LIN {X 0,Y 184.032,Z 367.437,A -85,B 0,C 180,E1 -22186.576,E2 -22186.576} C_VEL
LIN {X 0,Y 183.356,Z 367.135,A -85,B 0,C 180,E1 -22190.049,E2 -22190.049} C_VEL
LIN {X 0,Y 183.093,Z 365.736,A -85,B 0,C 180,E1 -22193.714,E2 -22193.714} C_VEL
LIN {X 0,Y 183.399,Z 363.047,A -85,B 0,C 180,E1 -22197.555,E2 -22197.555} C_VEL
LIN {X 0,Y 184.194,Z 359.068,A -85,B 0,C 180,E1 -22201.35,E2 -22201.35} C_VEL
LIN {X 0,Y 185.42,Z 353.009,A -85,B 0,C 180,E1 -22205.459,E2 -22205.459} C_VEL
LIN {X 0,Y 186.983,Z 346.449,A -85,B 0,C 180,E1 -22208.832,E2 -22208.832} C_VEL
LIN {X 0,Y 188.948,Z 338.257,A -85,B 0,C 180,E1 -22212.13,E2 -22212.13} C_VEL
LIN {X 0,Y 191.271,Z 328.831,A -85,B 0,C 180,E1 -22215.096,E2 -22215.096} C_VEL
LIN {X 0,Y 193.258,Z 319.749,A -85,B 0,C 180,E1 -22217.397,E2 -22217.397} C_VEL
LIN {X 0,Y 195.527,Z 308.58,A -85,B 0,C 180,E1 -22219.647,E2 -22219.647} C_VEL
LIN {X 0,Y 197.745,Z 296.151,A -85,B 0,C 180,E1 -22221.57,E2 -22221.57} C_VEL
LIN {X 0,Y 199.324,Z 284.381,A -85,B 0,C 180,E1 -22222.968,E2 -22222.968} C_VEL
LIN {X 0,Y 200.748,Z 270.755,A -85,B 0,C 180,E1 -22224.108,E2 -22224.108} C_VEL
LIN {X 0,Y 201.714,Z 257.362,A -85,B 0,C 180,E1 -22224.816,E2 -22224.816} C_VEL
LIN {X 0,Y 204.371,Z 205.343,A -85,B 0,C 180,E1 -22226.746,E2 -22226.746} C_VEL
LIN {X 0,Y 197.795,Z 189.738,A -85,B 0,C 180,E1 -22228.409,E2 -22228.409} C_VEL
LIN {X 0,Y 187.977,Z 169.046,A -85,B 0,C 180,E1 -22231.002,E2 -22231.002} C_VEL
LIN {X 0,Y 186.53,Z 166.516,A -85,B 0,C 180,E1 -22231.384,E2 -22231.384} C_VEL
LIN {X 0,Y 186.263,Z 165.286,A -85,B 0,C 180,E1 -22231.555,E2 -22231.555} C_VEL
LIN {X 0,Y 185.974,Z 165.321,A -85,B 0,C 180,E1 -22238.694,E2 -22238.694} C_VEL
LIN {X 0,Y 185.717,Z 165.352,A -85,B 0,C 180,E1 -22243.124,E2 -22243.124} C_VEL
LIN {X 0,Y 185.656,Z 165.356,A -85,B 0,C 180,E1 -22247.628,E2 -22247.628} C_VEL
LIN {X 0,Y 185.574,Z 165.367,A -85,B 0,C 180,E1 -22252.254,E2 -22252.254} C_VEL
LIN {X 0,Y 185.56,Z 165.368,A -85,B 0,C 180,E1 -22257.032,E2 -22257.032} C_VEL
LIN {X 0,Y 185.579,Z 165.367,A -85,B 0,C 180,E1 -22259.493,E2 -22259.493} C_VEL
LIN {X 0,Y 185.499,Z 165.377,A -85,B 0,C 180,E1 -22264.632,E2 -22264.632} C_VEL
LIN {X 0,Y 185.505,Z 165.377,A -85,B 0,C 180,E1 -22267.313,E2 -22267.313} C_VEL
LIN {X 0,Y 185.47,Z 165.369,A -85,B 0,C 180,E1 -22270.725,E2 -22270.725} C_VEL
LIN {X 0,Y 185.459,Z 165.384,A -85,B 0,C 180,E1 -22276.055,E2 -22276.055} C_VEL
LIN {X 0,Y 185.487,Z 165.365,A -85,B 0,C 180,E1 -22279.901,E2 -22279.901} C_VEL
LIN {X 0,Y 185.543,Z 165.368,A -85,B 0,C 180,E1 -22282.696,E2 -22282.696} C_VEL
LIN {X 0,Y 185.54,Z 165.366,A -85,B 0,C 180,E1 -22287.975,E2 -22287.975} C_VEL
LIN {X 0,Y 185.58,Z 165.348,A -85,B 0,C 180,E1 -22290.577,E2 -22290.577} C_VEL
LIN {X 0,Y 185.579,Z 165.367,A -85,B 0,C 180,E1 -22295.382,E2 -22295.382} C_VEL
LIN {X 0,Y 185.673,Z 165.341,A -85,B 0,C 180,E1 -22301.135,E2 -22301.135} C_VEL
LIN {X 0,Y 185.724,Z 165.342,A -85,B 0,C 180,E1 -22304.64,E2 -22304.64} C_VEL
LIN {X 0,Y 185.924,Z 165.323,A -85,B 0,C 180,E1 -22309.359,E2 -22309.359} C_VEL
LIN {X 0,Y 185.961,Z 165.303,A -85,B 0,C 180,E1 -22313.49,E2 -22313.49} C_VEL
LIN {X 0,Y 186.208,Z 165.286,A -85,B 0,C 180,E1 -22317.837,E2 -22317.837} C_VEL
LIN {X 0,Y 186.407,Z 165.26,A -85,B 0,C 180,E1 -22320,E2 -22320} C_VEL
LIN {X 0,Y 185.923,Z 165.31,A -85,B 0,C 180,E1 -22324.336,E2 -22324.336} C_VEL
LIN {X 0,Y 186.009,Z 165.314,A -85,B 0,C 180,E1 -22328.693,E2 -22328.693} C_VEL
LIN {X 0,Y 185.765,Z 165.335,A -85,B 0,C 180,E1 -22333.121,E2 -22333.121} C_VEL
LIN {X 0,Y 185.69,Z 165.353,A -85,B 0,C 180,E1 -22337.625,E2 -22337.625} C_VEL
LIN {X 0,Y 185.579,Z 165.366,A -85,B 0,C 180,E1 -22342.254,E2 -22342.254} C_VEL
LIN {X 0,Y 185.561,Z 165.365,A -85,B 0,C 180,E1 -22347.033,E2 -22347.033} C_VEL
LIN {X 0,Y 185.58,Z 165.369,A -85,B 0,C 180,E1 -22349.493,E2 -22349.493} C_VEL
LIN {X 0,Y 185.52,Z 165.377,A -85,B 0,C 180,E1 -22354.628,E2 -22354.628} C_VEL
LIN {X 0,Y 185.545,Z 165.372,A -85,B 0,C 180,E1 -22357.304,E2 -22357.304} C_VEL
LIN {X 0,Y 185.504,Z 165.379,A -85,B 0,C 180,E1 -22360.737,E2 -22360.737} C_VEL
LIN {X 0,Y 185.519,Z 165.377,A -85,B 0,C 180,E1 -22366.037,E2 -22366.037} C_VEL
LIN {X 0,Y 185.542,Z 165.525,A -85,B 0,C 180,E1 -22366.821,E2 -22366.821} C_VEL
LIN {X 0,Y 187.738,Z 174.486,A -85,B 0,C 180,E1 -22371.323,E2 -22371.323} C_VEL
LIN {X 0,Y 196.018,Z 195.049,A -85,B 0,C 180,E1 -22373.668,E2 -22373.668} C_VEL
LIN {X 0,Y 199.664,Z 205.529,A -85,B 0,C 180,E1 -22374.697,E2 -22374.697} C_VEL
LIN {X 0,Y 202.857,Z 235.414,A -85,B 0,C 180,E1 -22376.487,E2 -22376.487} C_VEL
LIN {X 0,Y 202.626,Z 245.83,A -85,B 0,C 180,E1 -22376.916,E2 -22376.916} C_VEL
LIN {X 0,Y 202.405,Z 251.4,A -85,B 0,C 180,E1 -22377.132,E2 -22377.132} C_VEL
LIN {X 0,Y 201.656,Z 257.229,A -85,B 0,C 180,E1 -22377.285,E2 -22377.285} C_VEL
LIN {X 0,Y 198.546,Z 266.659,A -85,B 0,C 180,E1 -22377.284,E2 -22377.284} C_VEL
LIN {X 0,Y 195.295,Z 276.077,A -85,B 0,C 180,E1 -22377.291,E2 -22377.291} C_VEL
LIN {X 0,Y 194.336,Z 281.893,A -85,B 0,C 180,E1 -22377.468,E2 -22377.468} C_VEL
LIN {X 0,Y 193.33,Z 293.632,A -85,B 0,C 180,E1 -22378.19,E2 -22378.19} C_VEL
LIN {X 0,Y 191.752,Z 305.726,A -85,B 0,C 180,E1 -22379.281,E2 -22379.281} C_VEL
LIN {X 0,Y 189.786,Z 316.758,A -85,B 0,C 180,E1 -22380.616,E2 -22380.616} C_VEL
LIN {X 0,Y 187.216,Z 329.252,A -85,B 0,C 180,E1 -22382.622,E2 -22382.622} C_VEL
LIN {X 0,Y 184.684,Z 340.28,A -85,B 0,C 180,E1 -22384.954,E2 -22384.954} C_VEL
LIN {X 0,Y 182.202,Z 350.699,A -85,B 0,C 180,E1 -22387.782,E2 -22387.782} C_VEL
LIN {X 0,Y 180.484,Z 357.527,A -85,B 0,C 180,E1 -22390.079,E2 -22390.079} C_VEL
LIN {X 0,Y 178.673,Z 365.629,A -85,B 0,C 180,E1 -22393.431,E2 -22393.431} C_VEL
LIN {X 0,Y 177.448,Z 371.066,A -85,B 0,C 180,E1 -22396.253,E2 -22396.253} C_VEL
LIN {X 0,Y 176.647,Z 376.382,A -85,B 0,C 180,E1 -22399.686,E2 -22399.686} C_VEL
LIN {X 0,Y 176.33,Z 380.466,A -85,B 0,C 180,E1 -22403.133,E2 -22403.133} C_VEL
LIN {X 0,Y 176.351,Z 382.551,A -85,B 0,C 180,E1 -22405.428,E2 -22405.428} C_VEL
LIN {X 0,Y 176.404,Z 384.172,A -85,B 0,C 180,E1 -22407.717,E2 -22407.717} C_VEL
LIN {X 0,Y 176.485,Z 385.363,A -85,B 0,C 180,E1 -22410,E2 -22410} C_VEL
LIN {X 0,Y 176.309,Z 386.103,A -85,B 0,C 180,E1 -22412.284,E2 -22412.284} C_VEL
LIN {X 0,Y 176.145,Z 386.398,A -85,B 0,C 180,E1 -22414.577,E2 -22414.577} C_VEL
LIN {X 0,Y 176.371,Z 385.833,A -85,B 0,C 180,E1 -22419.171,E2 -22419.171} C_VEL
LIN {X 0,Y 176.852,Z 384.98,A -85,B 0,C 180,E1 -22421.461,E2 -22421.461} C_VEL
LIN {X 0,Y 178.535,Z 382.023,A -85,B 0,C 180,E1 -22425.995,E2 -22425.995} C_VEL
LIN {X 0,Y 180.694,Z 378.736,A -85,B 0,C 180,E1 -22429.305,E2 -22429.305} C_VEL
LIN {X 0,Y 183.399,Z 374.424,A -85,B 0,C 180,E1 -22432.532,E2 -22432.532} C_VEL
LIN {X 0,Y 187.159,Z 367.956,A -85,B 0,C 180,E1 -22436.182,E2 -22436.182} C_VEL
LIN {X 0,Y 191.107,Z 360.986,A -85,B 0,C 180,E1 -22439.161,E2 -22439.161} C_VEL
LIN {X 0,Y 195.635,Z 352.395,A -85,B 0,C 180,E1 -22441.997,E2 -22441.997} C_VEL
LIN {X 0,Y 199.979,Z 343.651,A -85,B 0,C 180,E1 -22444.215,E2 -22444.215} C_VEL
LIN {X 0,Y 204.06,Z 334.168,A -85,B 0,C 180,E1 -22446.142,E2 -22446.142} C_VEL
LIN {X 0,Y 208.011,Z 323.894,A -85,B 0,C 180,E1 -22447.762,E2 -22447.762} C_VEL
LIN {X 0,Y 211.57,Z 312.785,A -85,B 0,C 180,E1 -22449.134,E2 -22449.134} C_VEL
LIN {X 0,Y 214.827,Z 300.374,A -85,B 0,C 180,E1 -22450.249,E2 -22450.249} C_VEL
LIN {X 0,Y 217.351,Z 286.914,A -85,B 0,C 180,E1 -22451.126,E2 -22451.126} C_VEL
LIN {X 0,Y 218.947,Z 273.192,A -85,B 0,C 180,E1 -22451.698,E2 -22451.698} C_VEL
LIN {X 0,Y 221.305,Z 243.676,A -85,B 0,C 180,E1 -22452.714,E2 -22452.714} C_VEL
LIN {X 0,Y 220.723,Z 234.505,A -85,B 0,C 180,E1 -22453.502,E2 -22453.502} C_VEL
LIN {X 0,Y 216.604,Z 223.631,A -85,B 0,C 180,E1 -22455.788,E2 -22455.788} C_VEL
LIN {X 0,Y 212.688,Z 215.258,A -85,B 0,C 180,E1 -22458.109,E2 -22458.109} C_VEL
LIN {X 0,Y 209.577,Z 209.321,A -85,B 0,C 180,E1 -22460.11,E2 -22460.11} C_VEL
LIN {X 0,Y 207.305,Z 205.119,A -85,B 0,C 180,E1 -22461.75,E2 -22461.75} C_VEL
LIN {X 0,Y 204.342,Z 199.923,A -85,B 0,C 180,E1 -22464.107,E2 -22464.107} C_VEL
LIN {X 0,Y 200.97,Z 194.246,A -85,B 0,C 180,E1 -22467.349,E2 -22467.349} C_VEL
LIN {X 0,Y 196.57,Z 187.167,A -85,B 0,C 180,E1 -22473.357,E2 -22473.357} C_VEL
LIN {X 0,Y 194.473,Z 184.049,A -85,B 0,C 180,E1 -22479.652,E2 -22479.652} C_VEL
LIN {X 0,Y 194.709,Z 184.022,A -85,B 0,C 180,E1 -22485.364,E2 -22485.364} C_VEL
LIN {X 0,Y 196.216,Z 184.626,A -85,B 0,C 180,E1 -22489.292,E2 -22489.292} C_VEL
LIN {X 0,Y 197.724,Z 187.889,A -85,B 0,C 180,E1 -22492.253,E2 -22492.253} C_VEL
LIN {X 0,Y 200.136,Z 189.87,A -85,B 0,C 180,E1 -22495.215,E2 -22495.215} C_VEL
LIN {X 0,Y 200.777,Z 190.672,A -85,B 0,C 180,E1 -22495.922,E2 -22495.922} C_VEL
LIN {X 0,Y 203.022,Z 193.797,A -85,B 0,C 180,E1 -22498.147,E2 -22498.147} C_VEL
LIN {X 0,Y 203.994,Z 195.111,A -85,B 0,C 180,E1 -22499.022,E2 -22499.022} C_VEL
LIN {X 0,Y 206.507,Z 198.84,A -85,B 0,C 180,E1 -22501.071,E2 -22501.071} C_VEL
LIN {X 0,Y 210.473,Z 204.645,A -85,B 0,C 180,E1 -22503.865,E2 -22503.865} C_VEL
LIN {X 0,Y 214.841,Z 211.746,A -85,B 0,C 180,E1 -22506.499,E2 -22506.499} C_VEL
LIN {X 0,Y 219.364,Z 219.717,A -85,B 0,C 180,E1 -22508.927,E2 -22508.927} C_VEL
LIN {X 0,Y 222.627,Z 226.3,A -85,B 0,C 180,E1 -22510.552,E2 -22510.552} C_VEL
LIN {X 0,Y 219.091,Z 267.39,A -85,B 0,C 180,E1 -22511.994,E2 -22511.994} C_VEL
LIN {X 0,Y 217.001,Z 281.249,A -85,B 0,C 180,E1 -22512.82,E2 -22512.82} C_VEL
LIN {X 0,Y 214.473,Z 293.514,A -85,B 0,C 180,E1 -22513.926,E2 -22513.926} C_VEL
LIN {X 0,Y 211.106,Z 305.921,A -85,B 0,C 180,E1 -22515.446,E2 -22515.446} C_VEL
LIN {X 0,Y 207.644,Z 316.071,A -85,B 0,C 180,E1 -22517.03,E2 -22517.03} C_VEL
LIN {X 0,Y 203.566,Z 326.285,A -85,B 0,C 180,E1 -22519.074,E2 -22519.074} C_VEL
LIN {X 0,Y 199.211,Z 335.653,A -85,B 0,C 180,E1 -22521.49,E2 -22521.49} C_VEL
LIN {X 0,Y 194.694,Z 344.181,A -85,B 0,C 180,E1 -22524.314,E2 -22524.314} C_VEL
LIN {X 0,Y 190.253,Z 351.606,A -85,B 0,C 180,E1 -22527.556,E2 -22527.556} C_VEL
LIN {X 0,Y 186.095,Z 357.882,A -85,B 0,C 180,E1 -22531.255,E2 -22531.255} C_VEL
LIN {X 0,Y 183.362,Z 361.587,A -85,B 0,C 180,E1 -22534.231,E2 -22534.231} C_VEL
LIN {X 0,Y 180.342,Z 365.302,A -85,B 0,C 180,E1 -22538.573,E2 -22538.573} C_VEL
LIN {X 0,Y 178.539,Z 367.039,A -85,B 0,C 180,E1 -22542.004,E2 -22542.004} C_VEL
LIN {X 0,Y 177.177,Z 367.836,A -85,B 0,C 180,E1 -22545.56,E2 -22545.56} C_VEL
LIN {X 0,Y 176.375,Z 367.638,A -85,B 0,C 180,E1 -22549.208,E2 -22549.208} C_VEL
LIN {X 0,Y 176.004,Z 366.246,A -85,B 0,C 180,E1 -22553.205,E2 -22553.205} C_VEL
LIN {X 0,Y 176.195,Z 363.867,A -85,B 0,C 180,E1 -22556.891,E2 -22556.891} C_VEL
LIN {X 0,Y 176.985,Z 359.996,A -85,B 0,C 180,E1 -22560.88,E2 -22560.88} C_VEL
LIN {X 0,Y 177.881,Z 355.57,A -85,B 0,C 180,E1 -22564.24,E2 -22564.24} C_VEL
LIN {X 0,Y 179.467,Z 348.824,A -85,B 0,C 180,E1 -22568.16,E2 -22568.16} C_VEL
LIN {X 0,Y 181.225,Z 341.748,A -85,B 0,C 180,E1 -22571.341,E2 -22571.341} C_VEL
LIN {X 0,Y 183.394,Z 333.098,A -85,B 0,C 180,E1 -22574.44,E2 -22574.44} C_VEL
LIN {X 0,Y 185.765,Z 323.252,A -85,B 0,C 180,E1 -22577.242,E2 -22577.242} C_VEL
LIN {X 0,Y 188.293,Z 311.74,A -85,B 0,C 180,E1 -22579.788,E2 -22579.788} C_VEL
LIN {X 0,Y 190.52,Z 300.077,A -85,B 0,C 180,E1 -22581.799,E2 -22581.799} C_VEL
LIN {X 0,Y 192.302,Z 288.407,A -85,B 0,C 180,E1 -22583.337,E2 -22583.337} C_VEL
LIN {X 0,Y 193.911,Z 274.589,A -85,B 0,C 180,E1 -22584.671,E2 -22584.671} C_VEL
LIN {X 0,Y 195.004,Z 261.627,A -85,B 0,C 180,E1 -22585.478,E2 -22585.478} C_VEL
LIN {X 0,Y 197.86,Z 206.871,A -85,B 0,C 180,E1 -22587.608,E2 -22587.608} C_VEL
LIN {X 0,Y 191.853,Z 192.642,A -85,B 0,C 180,E1 -22589.197,E2 -22589.197} C_VEL
LIN {X 0,Y 182.808,Z 173.416,A -85,B 0,C 180,E1 -22591.711,E2 -22591.711} C_VEL
LIN {X 0,Y 180.157,Z 169.113,A -85,B 0,C 180,E1 -22592.429,E2 -22592.429} C_VEL
LIN {X 0,Y 179.041,Z 166.186,A -85,B 0,C 180,E1 -22592.813,E2 -22592.813} C_VEL
LIN {X 0,Y 178.905,Z 166.204,A -85,B 0,C 180,E1 -22599.041,E2 -22599.041} C_VEL
LIN {X 0,Y 178.644,Z 166.233,A -85,B 0,C 180,E1 -22603.653,E2 -22603.653} C_VEL
LIN {X 0,Y 178.59,Z 166.239,A -85,B 0,C 180,E1 -22609.186,E2 -22609.186} C_VEL
LIN {X 0,Y 178.519,Z 166.247,A -85,B 0,C 180,E1 -22615.114,E2 -22615.114} C_VEL
LIN {X 0,Y 178.523,Z 166.246,A -85,B 0,C 180,E1 -22619.994,E2 -22619.994} C_VEL
LIN {X 0,Y 178.485,Z 166.252,A -85,B 0,C 180,E1 -22624.22,E2 -22624.22} C_VEL
LIN {X 0,Y 178.395,Z 166.258,A -85,B 0,C 180,E1 -22629.075,E2 -22629.075} C_VEL
LIN {X 0,Y 178.397,Z 166.251,A -85,B 0,C 180,E1 -22632.045,E2 -22632.045} C_VEL
LIN {X 0,Y 178.393,Z 166.262,A -85,B 0,C 180,E1 -22635.164,E2 -22635.164} C_VEL
LIN {X 0,Y 178.409,Z 166.252,A -85,B 0,C 180,E1 -22638.457,E2 -22638.457} C_VEL
LIN {X 0,Y 178.463,Z 166.243,A -85,B 0,C 180,E1 -22641.963,E2 -22641.963} C_VEL
LIN {X 0,Y 178.489,Z 166.248,A -85,B 0,C 180,E1 -22646.548,E2 -22646.548} C_VEL
LIN {X 0,Y 178.521,Z 166.229,A -85,B 0,C 180,E1 -22650.008,E2 -22650.008} C_VEL
LIN {X 0,Y 178.519,Z 166.245,A -85,B 0,C 180,E1 -22654.886,E2 -22654.886} C_VEL
LIN {X 0,Y 178.621,Z 166.221,A -85,B 0,C 180,E1 -22660.786,E2 -22660.786} C_VEL
LIN {X 0,Y 178.665,Z 166.218,A -85,B 0,C 180,E1 -22664.017,E2 -22664.017} C_VEL
LIN {X 0,Y 178.861,Z 166.203,A -85,B 0,C 180,E1 -22669.211,E2 -22669.211} C_VEL
LIN {X 0,Y 178.925,Z 166.178,A -85,B 0,C 180,E1 -22673.233,E2 -22673.233} C_VEL
LIN {X 0,Y 179.154,Z 166.165,A -85,B 0,C 180,E1 -22677.752,E2 -22677.752} C_VEL
LIN {X 0,Y 179.37,Z 166.137,A -85,B 0,C 180,E1 -22680,E2 -22680} C_VEL
LIN {X 0,Y 178.871,Z 166.189,A -85,B 0,C 180,E1 -22684.508,E2 -22684.508} C_VEL
LIN {X 0,Y 178.96,Z 166.191,A -85,B 0,C 180,E1 -22689.038,E2 -22689.038} C_VEL
LIN {X 0,Y 178.687,Z 166.219,A -85,B 0,C 180,E1 -22693.65,E2 -22693.65} C_VEL
LIN {X 0,Y 178.649,Z 166.229,A -85,B 0,C 180,E1 -22698.344,E2 -22698.344} C_VEL
LIN {X 0,Y 178.498,Z 166.25,A -85,B 0,C 180,E1 -22703.187,E2 -22703.187} C_VEL
LIN {X 0,Y 178.487,Z 166.25,A -85,B 0,C 180,E1 -22708.198,E2 -22708.198} C_VEL
LIN {X 0,Y 178.48,Z 166.252,A -85,B 0,C 180,E1 -22710.791,E2 -22710.791} C_VEL
LIN {X 0,Y 178.497,Z 166.253,A -85,B 0,C 180,E1 -22714.225,E2 -22714.225} C_VEL
LIN {X 0,Y 178.427,Z 166.258,A -85,B 0,C 180,E1 -22719.067,E2 -22719.067} C_VEL
LIN {X 0,Y 178.433,Z 166.258,A -85,B 0,C 180,E1 -22722.036,E2 -22722.036} C_VEL
LIN {X 0,Y 178.497,Z 166.39,A -85,B 0,C 180,E1 -22725.937,E2 -22725.937} C_VEL
LIN {X 0,Y 180.402,Z 174.103,A -85,B 0,C 180,E1 -22729.974,E2 -22729.974} C_VEL
LIN {X 0,Y 187.223,Z 190.403,A -85,B 0,C 180,E1 -22732.028,E2 -22732.028} C_VEL
LIN {X 0,Y 193.54,Z 207.992,A -85,B 0,C 180,E1 -22733.898,E2 -22733.898} C_VEL
LIN {X 0,Y 196.515,Z 237.335,A -85,B 0,C 180,E1 -22735.695,E2 -22735.695} C_VEL
LIN {X 0,Y 194.646,Z 277.657,A -85,B 0,C 180,E1 -22737.285,E2 -22737.285} C_VEL
LIN {X 0,Y 194.336,Z 281.893,A -85,B 0,C 180,E1 -22737.468,E2 -22737.468} C_VEL
LIN {X 0,Y 193.328,Z 287.66,A -85,B 0,C 180,E1 -22737.702,E2 -22737.702} C_VEL
LIN {X 0,Y 189.715,Z 296.836,A -85,B 0,C 180,E1 -22738.027,E2 -22738.027} C_VEL
LIN {X 0,Y 185.718,Z 305.78,A -85,B 0,C 180,E1 -22738.565,E2 -22738.565} C_VEL
LIN {X 0,Y 184.127,Z 311.192,A -85,B 0,C 180,E1 -22739.133,E2 -22739.133} C_VEL
LIN {X 0,Y 181.892,Z 322.677,A -85,B 0,C 180,E1 -22740.803,E2 -22740.803} C_VEL
LIN {X 0,Y 179.366,Z 333.828,A -85,B 0,C 180,E1 -22742.903,E2 -22742.903} C_VEL
LIN {X 0,Y 176.898,Z 343.897,A -85,B 0,C 180,E1 -22745.345,E2 -22745.345} C_VEL
LIN {X 0,Y 174.598,Z 352.705,A -85,B 0,C 180,E1 -22748.021,E2 -22748.021} C_VEL
LIN {X 0,Y 172.691,Z 360.577,A -85,B 0,C 180,E1 -22751,E2 -22751} C_VEL
LIN {X 0,Y 171.016,Z 367.975,A -85,B 0,C 180,E1 -22754.507,E2 -22754.507} C_VEL
LIN {X 0,Y 169.885,Z 373.858,A -85,B 0,C 180,E1 -22758.062,E2 -22758.062} C_VEL
LIN {X 0,Y 169.342,Z 378.447,A -85,B 0,C 180,E1 -22761.648,E2 -22761.648} C_VEL
LIN {X 0,Y 169.298,Z 381.892,A -85,B 0,C 180,E1 -22765.237,E2 -22765.237} C_VEL
LIN {X 0,Y 169.321,Z 383.563,A -85,B 0,C 180,E1 -22767.621,E2 -22767.621} C_VEL
LIN {X 0,Y 169.419,Z 384.804,A -85,B 0,C 180,E1 -22770,E2 -22770} C_VEL
LIN {X 0,Y 169.103,Z 385.901,A -85,B 0,C 180,E1 -22774.084,E2 -22774.084} C_VEL
LIN {X 0,Y 169.082,Z 385.934,A -85,B 0,C 180,E1 -22777.163,E2 -22777.163} C_VEL
LIN {X 0,Y 169.847,Z 384.711,A -85,B 0,C 180,E1 -22781.94,E2 -22781.94} C_VEL
LIN {X 0,Y 170.592,Z 383.529,A -85,B 0,C 180,E1 -22784.311,E2 -22784.311} C_VEL
LIN {X 0,Y 172.402,Z 380.967,A -85,B 0,C 180,E1 -22787.802,E2 -22787.802} C_VEL
LIN {X 0,Y 174.804,Z 377.447,A -85,B 0,C 180,E1 -22791.213,E2 -22791.213} C_VEL
LIN {X 0,Y 178.323,Z 372.169,A -85,B 0,C 180,E1 -22794.977,E2 -22794.977} C_VEL
LIN {X 0,Y 182.754,Z 365.018,A -85,B 0,C 180,E1 -22798.731,E2 -22798.731} C_VEL
LIN {X 0,Y 187.314,Z 357.486,A -85,B 0,C 180,E1 -22801.687,E2 -22801.687} C_VEL
LIN {X 0,Y 191.489,Z 349.874,A -85,B 0,C 180,E1 -22804.035,E2 -22804.035} C_VEL
LIN {X 0,Y 196.485,Z 339.699,A -85,B 0,C 180,E1 -22806.487,E2 -22806.487} C_VEL
LIN {X 0,Y 201.442,Z 328.132,A -85,B 0,C 180,E1 -22808.581,E2 -22808.581} C_VEL
LIN {X 0,Y 205.643,Z 316.541,A -85,B 0,C 180,E1 -22810.17,E2 -22810.17} C_VEL
LIN {X 0,Y 209.262,Z 304.386,A -85,B 0,C 180,E1 -22811.391,E2 -22811.391} C_VEL
LIN {X 0,Y 212.354,Z 290.559,A -85,B 0,C 180,E1 -22812.4,E2 -22812.4} C_VEL
LIN {X 0,Y 214.316,Z 276.784,A -85,B 0,C 180,E1 -22813.058,E2 -22813.058} C_VEL
LIN {X 0,Y 217.022,Z 244.728,A -85,B 0,C 180,E1 -22814.194,E2 -22814.194} C_VEL
LIN {X 0,Y 216.568,Z 237.513,A -85,B 0,C 180,E1 -22814.852,E2 -22814.852} C_VEL
LIN {X 0,Y 212.945,Z 227.818,A -85,B 0,C 180,E1 -22817.03,E2 -22817.03} C_VEL
LIN {X 0,Y 209.267,Z 219.693,A -85,B 0,C 180,E1 -22819.399,E2 -22819.399} C_VEL
LIN {X 0,Y 206.901,Z 214.908,A -85,B 0,C 180,E1 -22821.071,E2 -22821.071} C_VEL
LIN {X 0,Y 204.936,Z 211.064,A -85,B 0,C 180,E1 -22822.595,E2 -22822.595} C_VEL
LIN {X 0,Y 202.228,Z 206.106,A -85,B 0,C 180,E1 -22824.903,E2 -22824.903} C_VEL
LIN {X 0,Y 199.176,Z 200.711,A -85,B 0,C 180,E1 -22828.042,E2 -22828.042} C_VEL
LIN {X 0,Y 195.434,Z 194.14,A -85,B 0,C 180,E1 -22833.527,E2 -22833.527} C_VEL
LIN {X 0,Y 193.42,Z 190.997,A -85,B 0,C 180,E1 -22839.911,E2 -22839.911} C_VEL
LIN {X 0,Y 193.667,Z 191.042,A -85,B 0,C 180,E1 -22845.284,E2 -22845.284} C_VEL
LIN {X 0,Y 195.007,Z 191.628,A -85,B 0,C 180,E1 -22848.961,E2 -22848.961} C_VEL
LIN {X 0,Y 196.459,Z 194.834,A -85,B 0,C 180,E1 -22851.98,E2 -22851.98} C_VEL
LIN {X 0,Y 199.006,Z 197.071,A -85,B 0,C 180,E1 -22855.188,E2 -22855.188} C_VEL
LIN {X 0,Y 201.341,Z 200.469,A -85,B 0,C 180,E1 -22857.65,E2 -22857.65} C_VEL
LIN {X 0,Y 202.35,Z 202.107,A -85,B 0,C 180,E1 -22858.621,E2 -22858.621} C_VEL
LIN {X 0,Y 205.587,Z 206.99,A -85,B 0,C 180,E1 -22861.309,E2 -22861.309} C_VEL
LIN {X 0,Y 208.415,Z 211.334,A -85,B 0,C 180,E1 -22863.346,E2 -22863.346} C_VEL
LIN {X 0,Y 213.522,Z 220.044,A -85,B 0,C 180,E1 -22866.539,E2 -22866.539} C_VEL
LIN {X 0,Y 217.995,Z 228.789,A -85,B 0,C 180,E1 -22869.013,E2 -22869.013} C_VEL
LIN {X 0,Y 218.226,Z 229.297,A -85,B 0,C 180,E1 -22869.135,E2 -22869.135} C_VEL
LIN {X 0,Y 214.818,Z 267.651,A -85,B 0,C 180,E1 -22870.5,E2 -22870.5} C_VEL
LIN {X 0,Y 212.708,Z 281.185,A -85,B 0,C 180,E1 -22871.302,E2 -22871.302} C_VEL
LIN {X 0,Y 209.874,Z 294.213,A -85,B 0,C 180,E1 -22872.479,E2 -22872.479} C_VEL
LIN {X 0,Y 206.349,Z 306.542,A -85,B 0,C 180,E1 -22874.015,E2 -22874.015} C_VEL
LIN {X 0,Y 202.36,Z 317.541,A -85,B 0,C 180,E1 -22875.77,E2 -22875.77} C_VEL
LIN {X 0,Y 198.123,Z 327.457,A -85,B 0,C 180,E1 -22877.823,E2 -22877.823} C_VEL
LIN {X 0,Y 193.467,Z 336.894,A -85,B 0,C 180,E1 -22880.332,E2 -22880.332} C_VEL
LIN {X 0,Y 189.139,Z 344.578,A -85,B 0,C 180,E1 -22882.942,E2 -22882.942} C_VEL
LIN {X 0,Y 185.246,Z 350.857,A -85,B 0,C 180,E1 -22885.679,E2 -22885.679} C_VEL
LIN {X 0,Y 180.991,Z 356.912,A -85,B 0,C 180,E1 -22889.111,E2 -22889.111} C_VEL
LIN {X 0,Y 178.021,Z 360.774,A -85,B 0,C 180,E1 -22892,E2 -22892} C_VEL
LIN {X 0,Y 175.409,Z 363.888,A -85,B 0,C 180,E1 -22895.123,E2 -22895.123} C_VEL
LIN {X 0,Y 172.696,Z 366.692,A -85,B 0,C 180,E1 -22899.357,E2 -22899.357} C_VEL
LIN {X 0,Y 171.245,Z 367.811,A -85,B 0,C 180,E1 -22902.377,E2 -22902.377} C_VEL
LIN {X 0,Y 170.119,Z 368.261,A -85,B 0,C 180,E1 -22905.388,E2 -22905.388} C_VEL
LIN {X 0,Y 169.406,Z 368.094,A -85,B 0,C 180,E1 -22908.412,E2 -22908.412} C_VEL
LIN {X 0,Y 168.938,Z 366.95,A -85,B 0,C 180,E1 -22912.224,E2 -22912.224} C_VEL
LIN {X 0,Y 169.029,Z 364.612,A -85,B 0,C 180,E1 -22916.26,E2 -22916.26} C_VEL
LIN {X 0,Y 169.762,Z 360.908,A -85,B 0,C 180,E1 -22920.386,E2 -22920.386} C_VEL
LIN {X 0,Y 170.68,Z 356.486,A -85,B 0,C 180,E1 -22923.989,E2 -22923.989} C_VEL
LIN {X 0,Y 172.129,Z 350.363,A -85,B 0,C 180,E1 -22927.81,E2 -22927.81} C_VEL
LIN {X 0,Y 173.862,Z 343.579,A -85,B 0,C 180,E1 -22931.133,E2 -22931.133} C_VEL
LIN {X 0,Y 176.095,Z 335.092,A -85,B 0,C 180,E1 -22934.415,E2 -22934.415} C_VEL
LIN {X 0,Y 178.529,Z 325.323,A -85,B 0,C 180,E1 -22937.402,E2 -22937.402} C_VEL
LIN {X 0,Y 180.988,Z 314.836,A -85,B 0,C 180,E1 -22939.937,E2 -22939.937} C_VEL
LIN {X 0,Y 183.317,Z 303.541,A -85,B 0,C 180,E1 -22942.061,E2 -22942.061} C_VEL
LIN {X 0,Y 185.479,Z 290.97,A -85,B 0,C 180,E1 -22943.883,E2 -22943.883} C_VEL
LIN {X 0,Y 187.06,Z 278.487,A -85,B 0,C 180,E1 -22945.218,E2 -22945.218} C_VEL
LIN {X 0,Y 188.379,Z 264.652,A -85,B 0,C 180,E1 -22946.214,E2 -22946.214} C_VEL
LIN {X 0,Y 191.526,Z 208.863,A -85,B 0,C 180,E1 -22948.47,E2 -22948.47} C_VEL
LIN {X 0,Y 186.228,Z 196.209,A -85,B 0,C 180,E1 -22949.955,E2 -22949.955} C_VEL
LIN {X 0,Y 177.713,Z 177.9,A -85,B 0,C 180,E1 -22952.424,E2 -22952.424} C_VEL
LIN {X 0,Y 173.161,Z 170.297,A -85,B 0,C 180,E1 -22953.741,E2 -22953.741} C_VEL
LIN {X 0,Y 171.984,Z 167.796,A -85,B 0,C 180,E1 -22954.127,E2 -22954.127} C_VEL
LIN {X 0,Y 171.835,Z 167.083,A -85,B 0,C 180,E1 -22954.295,E2 -22954.295} C_VEL
LIN {X 0,Y 171.843,Z 167.082,A -85,B 0,C 180,E1 -22959.415,E2 -22959.415} C_VEL
LIN {X 0,Y 171.558,Z 167.116,A -85,B 0,C 180,E1 -22964.229,E2 -22964.229} C_VEL
LIN {X 0,Y 171.515,Z 167.119,A -85,B 0,C 180,E1 -22969.534,E2 -22969.534} C_VEL
LIN {X 0,Y 171.458,Z 167.126,A -85,B 0,C 180,E1 -22975.609,E2 -22975.609} C_VEL
LIN {X 0,Y 171.442,Z 167.128,A -85,B 0,C 180,E1 -22980.587,E2 -22980.587} C_VEL
LIN {X 0,Y 171.392,Z 167.134,A -85,B 0,C 180,E1 -22985.035,E2 -22985.035} C_VEL
LIN {X 0,Y 171.357,Z 167.135,A -85,B 0,C 180,E1 -22988.808,E2 -22988.808} C_VEL
LIN {X 0,Y 171.32,Z 167.142,A -85,B 0,C 180,E1 -22994.217,E2 -22994.217} C_VEL
LIN {X 0,Y 171.343,Z 167.131,A -85,B 0,C 180,E1 -22998.984,E2 -22998.984} C_VEL
LIN {X 0,Y 171.412,Z 167.121,A -85,B 0,C 180,E1 -23002.048,E2 -23002.048} C_VEL
LIN {X 0,Y 171.409,Z 167.131,A -85,B 0,C 180,E1 -23005.087,E2 -23005.087} C_VEL
LIN {X 0,Y 171.446,Z 167.107,A -85,B 0,C 180,E1 -23010.534,E2 -23010.534} C_VEL
LIN {X 0,Y 171.444,Z 167.13,A -85,B 0,C 180,E1 -23015.8,E2 -23015.8} C_VEL
LIN {X 0,Y 171.577,Z 167.097,A -85,B 0,C 180,E1 -23020.872,E2 -23020.872} C_VEL
LIN {X 0,Y 171.609,Z 167.105,A -85,B 0,C 180,E1 -23025.776,E2 -23025.776} C_VEL
LIN {X 0,Y 171.889,Z 167.068,A -85,B 0,C 180,E1 -23030.588,E2 -23030.588} C_VEL
LIN {X 0,Y 171.822,Z 167.068,A -85,B 0,C 180,E1 -23035.308,E2 -23035.308} C_VEL
LIN {X 0,Y 172.333,Z 167.013,A -85,B 0,C 180,E1 -23040.001,E2 -23040.001} C_VEL
LIN {X 0,Y 171.82,Z 167.067,A -85,B 0,C 180,E1 -23044.693,E2 -23044.693} C_VEL
LIN {X 0,Y 171.889,Z 167.07,A -85,B 0,C 180,E1 -23049.413,E2 -23049.413} C_VEL
LIN {X 0,Y 171.61,Z 167.101,A -85,B 0,C 180,E1 -23054.225,E2 -23054.225} C_VEL
LIN {X 0,Y 171.541,Z 167.109,A -85,B 0,C 180,E1 -23059.558,E2 -23059.558} C_VEL
LIN {X 0,Y 171.46,Z 167.123,A -85,B 0,C 180,E1 -23065.61,E2 -23065.61} C_VEL
LIN {X 0,Y 171.443,Z 167.129,A -85,B 0,C 180,E1 -23070.587,E2 -23070.587} C_VEL
LIN {X 0,Y 171.408,Z 167.134,A -85,B 0,C 180,E1 -23075.032,E2 -23075.032} C_VEL
LIN {X 0,Y 171.387,Z 167.135,A -85,B 0,C 180,E1 -23078.82,E2 -23078.82} C_VEL
LIN {X 0,Y 171.417,Z 167.131,A -85,B 0,C 180,E1 -23084.899,E2 -23084.899} C_VEL
LIN {X 0,Y 173.008,Z 173.62,A -85,B 0,C 180,E1 -23088.507,E2 -23088.507} C_VEL
LIN {X 0,Y 180.402,Z 190.875,A -85,B 0,C 180,E1 -23090.851,E2 -23090.851} C_VEL
LIN {X 0,Y 187.215,Z 209.276,A -85,B 0,C 180,E1 -23092.963,E2 -23092.963} C_VEL
LIN {X 0,Y 189.706,Z 233.597,A -85,B 0,C 180,E1 -23094.537,E2 -23094.537} C_VEL
LIN {X 0,Y 190.149,Z 239.469,A -85,B 0,C 180,E1 -23094.883,E2 -23094.883} C_VEL
LIN {X 0,Y 187.716,Z 283.904,A -85,B 0,C 180,E1 -23096.721,E2 -23096.721} C_VEL
LIN {X 0,Y 186.499,Z 295.587,A -85,B 0,C 180,E1 -23097.521,E2 -23097.521} C_VEL
LIN {X 0,Y 184.692,Z 308.172,A -85,B 0,C 180,E1 -23098.771,E2 -23098.771} C_VEL
LIN {X 0,Y 184.127,Z 311.192,A -85,B 0,C 180,E1 -23099.133,E2 -23099.133} C_VEL
LIN {X 0,Y 182.463,Z 316.588,A -85,B 0,C 180,E1 -23099.781,E2 -23099.781} C_VEL
LIN {X 0,Y 177.98,Z 324.89,A -85,B 0,C 180,E1 -23100.806,E2 -23100.806} C_VEL
LIN {X 0,Y 173.453,Z 332.743,A -85,B 0,C 180,E1 -23102.074,E2 -23102.074} C_VEL
LIN {X 0,Y 171.732,Z 337.396,A -85,B 0,C 180,E1 -23103.088,E2 -23103.088} C_VEL
LIN {X 0,Y 169.45,Z 346.282,A -85,B 0,C 180,E1 -23105.496,E2 -23105.496} C_VEL
LIN {X 0,Y 167.007,Z 354.911,A -85,B 0,C 180,E1 -23108.394,E2 -23108.394} C_VEL
LIN {X 0,Y 164.997,Z 363.343,A -85,B 0,C 180,E1 -23112.012,E2 -23112.012} C_VEL
LIN {X 0,Y 163.387,Z 370.08,A -85,B 0,C 180,E1 -23115.68,E2 -23115.68} C_VEL
LIN {X 0,Y 162.42,Z 376.201,A -85,B 0,C 180,E1 -23120.033,E2 -23120.033} C_VEL
LIN {X 0,Y 162.175,Z 380.127,A -85,B 0,C 180,E1 -23123.78,E2 -23123.78} C_VEL
LIN {X 0,Y 162.241,Z 382.95,A -85,B 0,C 180,E1 -23127.517,E2 -23127.517} C_VEL
LIN {X 0,Y 162.353,Z 384.24,A -85,B 0,C 180,E1 -23130,E2 -23130} C_VEL
LIN {X 0,Y 162.044,Z 385.395,A -85,B 0,C 180,E1 -23134.02,E2 -23134.02} C_VEL
LIN {X 0,Y 162.005,Z 385.563,A -85,B 0,C 180,E1 -23137.478,E2 -23137.478} C_VEL
LIN {X 0,Y 162.859,Z 384.444,A -85,B 0,C 180,E1 -23142.461,E2 -23142.461} C_VEL
LIN {X 0,Y 164.908,Z 381.804,A -85,B 0,C 180,E1 -23147.357,E2 -23147.357} C_VEL
LIN {X 0,Y 167.279,Z 378.731,A -85,B 0,C 180,E1 -23150.923,E2 -23150.923} C_VEL
LIN {X 0,Y 170.331,Z 374.668,A -85,B 0,C 180,E1 -23154.368,E2 -23154.368} C_VEL
LIN {X 0,Y 173.864,Z 369.525,A -85,B 0,C 180,E1 -23157.701,E2 -23157.701} C_VEL
LIN {X 0,Y 178.099,Z 363.146,A -85,B 0,C 180,E1 -23160.863,E2 -23160.863} C_VEL
LIN {X 0,Y 183.01,Z 355.242,A -85,B 0,C 180,E1 -23163.837,E2 -23163.837} C_VEL
LIN {X 0,Y 188.522,Z 345.501,A -85,B 0,C 180,E1 -23166.617,E2 -23166.617} C_VEL
LIN {X 0,Y 193.42,Z 335.554,A -85,B 0,C 180,E1 -23168.813,E2 -23168.813} C_VEL
LIN {X 0,Y 198.206,Z 324.402,A -85,B 0,C 180,E1 -23170.657,E2 -23170.657} C_VEL
LIN {X 0,Y 202.032,Z 313.662,A -85,B 0,C 180,E1 -23172.039,E2 -23172.039} C_VEL
LIN {X 0,Y 205.547,Z 301.925,A -85,B 0,C 180,E1 -23173.143,E2 -23173.143} C_VEL
LIN {X 0,Y 208.443,Z 288.661,A -85,B 0,C 180,E1 -23174.061,E2 -23174.061} C_VEL
LIN {X 0,Y 210.409,Z 274.561,A -85,B 0,C 180,E1 -23174.704,E2 -23174.704} C_VEL
LIN {X 0,Y 212.927,Z 245.798,A -85,B 0,C 180,E1 -23175.718,E2 -23175.718} C_VEL
LIN {X 0,Y 212.59,Z 240.826,A -85,B 0,C 180,E1 -23176.214,E2 -23176.214} C_VEL
LIN {X 0,Y 209.622,Z 232.429,A -85,B 0,C 180,E1 -23178.196,E2 -23178.196} C_VEL
LIN {X 0,Y 206.419,Z 225.083,A -85,B 0,C 180,E1 -23180.415,E2 -23180.415} C_VEL
LIN {X 0,Y 204.303,Z 220.503,A -85,B 0,C 180,E1 -23182.058,E2 -23182.058} C_VEL
LIN {X 0,Y 202.218,Z 216.36,A -85,B 0,C 180,E1 -23183.784,E2 -23183.784} C_VEL
LIN {X 0,Y 200.091,Z 212.133,A -85,B 0,C 180,E1 -23185.806,E2 -23185.806} C_VEL
LIN {X 0,Y 197.491,Z 207.293,A -85,B 0,C 180,E1 -23188.657,E2 -23188.657} C_VEL
LIN {X 0,Y 194.017,Z 200.846,A -85,B 0,C 180,E1 -23194.234,E2 -23194.234} C_VEL
LIN {X 0,Y 192.394,Z 198.091,A -85,B 0,C 180,E1 -23199.799,E2 -23199.799} C_VEL
LIN {X 0,Y 192.613,Z 198.056,A -85,B 0,C 180,E1 -23205.201,E2 -23205.201} C_VEL
LIN {X 0,Y 193.785,Z 198.59,A -85,B 0,C 180,E1 -23208.604,E2 -23208.604} C_VEL
LIN {X 0,Y 195.065,Z 201.598,A -85,B 0,C 180,E1 -23211.497,E2 -23211.497} C_VEL
LIN {X 0,Y 197.52,Z 203.922,A -85,B 0,C 180,E1 -23214.747,E2 -23214.747} C_VEL
LIN {X 0,Y 199.714,Z 207.184,A -85,B 0,C 180,E1 -23217.184,E2 -23217.184} C_VEL
LIN {X 0,Y 202.55,Z 211.782,A -85,B 0,C 180,E1 -23219.865,E2 -23219.865} C_VEL
LIN {X 0,Y 206.015,Z 217.377,A -85,B 0,C 180,E1 -23222.552,E2 -23222.552} C_VEL
LIN {X 0,Y 210.642,Z 225.641,A -85,B 0,C 180,E1 -23225.654,E2 -23225.654} C_VEL
LIN {X 0,Y 213.989,Z 232.426,A -85,B 0,C 180,E1 -23227.667,E2 -23227.667} C_VEL
LIN {X 0,Y 210.595,Z 268.734,A -85,B 0,C 180,E1 -23228.989,E2 -23228.989} C_VEL
LIN {X 0,Y 208.382,Z 282.156,A -85,B 0,C 180,E1 -23229.797,E2 -23229.797} C_VEL
LIN {X 0,Y 205.622,Z 294.324,A -85,B 0,C 180,E1 -23230.903,E2 -23230.903} C_VEL
LIN {X 0,Y 201.977,Z 306.532,A -85,B 0,C 180,E1 -23232.406,E2 -23232.406} C_VEL
LIN {X 0,Y 197.876,Z 317.509,A -85,B 0,C 180,E1 -23234.154,E2 -23234.154} C_VEL
LIN {X 0,Y 193.779,Z 326.749,A -85,B 0,C 180,E1 -23236.038,E2 -23236.038} C_VEL
LIN {X 0,Y 188.955,Z 336.098,A -85,B 0,C 180,E1 -23238.48,E2 -23238.48} C_VEL
LIN {X 0,Y 184.472,Z 343.744,A -85,B 0,C 180,E1 -23241.03,E2 -23241.03} C_VEL
LIN {X 0,Y 180.062,Z 350.502,A -85,B 0,C 180,E1 -23243.904,E2 -23243.904} C_VEL
LIN {X 0,Y 176.147,Z 355.861,A -85,B 0,C 180,E1 -23246.835,E2 -23246.835} C_VEL
LIN {X 0,Y 171.818,Z 361.243,A -85,B 0,C 180,E1 -23250.799,E2 -23250.799} C_VEL
LIN {X 0,Y 169.162,Z 364.154,A -85,B 0,C 180,E1 -23253.808,E2 -23253.808} C_VEL
LIN {X 0,Y 166.966,Z 366.315,A -85,B 0,C 180,E1 -23256.894,E2 -23256.894} C_VEL
LIN {X 0,Y 165.201,Z 367.786,A -85,B 0,C 180,E1 -23260.026,E2 -23260.026} C_VEL
LIN {X 0,Y 163.692,Z 368.569,A -85,B 0,C 180,E1 -23263.388,E2 -23263.388} C_VEL
LIN {X 0,Y 162.517,Z 368.555,A -85,B 0,C 180,E1 -23267.32,E2 -23267.32} C_VEL
LIN {X 0,Y 161.9,Z 367.499,A -85,B 0,C 180,E1 -23271.386,E2 -23271.386} C_VEL
LIN {X 0,Y 161.868,Z 365.257,A -85,B 0,C 180,E1 -23275.637,E2 -23275.637} C_VEL
LIN {X 0,Y 162.514,Z 361.763,A -85,B 0,C 180,E1 -23279.871,E2 -23279.871} C_VEL
LIN {X 0,Y 163.314,Z 358.119,A -85,B 0,C 180,E1 -23283.132,E2 -23283.132} C_VEL
LIN {X 0,Y 164.5,Z 353.02,A -85,B 0,C 180,E1 -23286.722,E2 -23286.722} C_VEL
LIN {X 0,Y 166.153,Z 346.725,A -85,B 0,C 180,E1 -23290.222,E2 -23290.222} C_VEL
LIN {X 0,Y 168.326,Z 338.543,A -85,B 0,C 180,E1 -23293.8,E2 -23293.8} C_VEL
LIN {X 0,Y 170.81,Z 329.511,A -85,B 0,C 180,E1 -23296.921,E2 -23296.921} C_VEL
LIN {X 0,Y 173.339,Z 319.066,A -85,B 0,C 180,E1 -23299.783,E2 -23299.783} C_VEL
LIN {X 0,Y 176.034,Z 307.201,A -85,B 0,C 180,E1 -23302.286,E2 -23302.286} C_VEL
LIN {X 0,Y 178.269,Z 295.416,A -85,B 0,C 180,E1 -23304.202,E2 -23304.202} C_VEL
LIN {X 0,Y 180.191,Z 282.123,A -85,B 0,C 180,E1 -23305.806,E2 -23305.806} C_VEL
LIN {X 0,Y 181.602,Z 268.977,A -85,B 0,C 180,E1 -23306.915,E2 -23306.915} C_VEL
LIN {X 0,Y 182.706,Z 252.516,A -85,B 0,C 180,E1 -23307.727,E2 -23307.727} C_VEL
LIN {X 0,Y 185.087,Z 210.463,A -85,B 0,C 180,E1 -23309.436,E2 -23309.436} C_VEL
LIN {X 0,Y 180.338,Z 199.108,A -85,B 0,C 180,E1 -23310.826,E2 -23310.826} C_VEL
LIN {X 0,Y 172.367,Z 181.822,A -85,B 0,C 180,E1 -23313.263,E2 -23313.263} C_VEL
LIN {X 0,Y 164.994,Z 169.121,A -85,B 0,C 180,E1 -23315.576,E2 -23315.576} C_VEL
LIN {X 0,Y 164.753,Z 167.965,A -85,B 0,C 180,E1 -23315.815,E2 -23315.815} C_VEL
LIN {X 0,Y 164.764,Z 167.963,A -85,B 0,C 180,E1 -23319.824,E2 -23319.824} C_VEL
LIN {X 0,Y 164.486,Z 167.996,A -85,B 0,C 180,E1 -23324.854,E2 -23324.854} C_VEL
LIN {X 0,Y 164.449,Z 167.999,A -85,B 0,C 180,E1 -23329.992,E2 -23329.992} C_VEL
LIN {X 0,Y 164.385,Z 168.007,A -85,B 0,C 180,E1 -23336.129,E2 -23336.129} C_VEL
LIN {X 0,Y 164.375,Z 168.007,A -85,B 0,C 180,E1 -23341.228,E2 -23341.228} C_VEL
LIN {X 0,Y 164.294,Z 168.02,A -85,B 0,C 180,E1 -23346.789,E2 -23346.789} C_VEL
LIN {X 0,Y 164.29,Z 168.01,A -85,B 0,C 180,E1 -23349.916,E2 -23349.916} C_VEL
LIN {X 0,Y 164.278,Z 168.017,A -85,B 0,C 180,E1 -23353.342,E2 -23353.342} C_VEL
LIN {X 0,Y 164.291,Z 168.017,A -85,B 0,C 180,E1 -23356.809,E2 -23356.809} C_VEL
LIN {X 0,Y 164.304,Z 168.001,A -85,B 0,C 180,E1 -23360.348,E2 -23360.348} C_VEL
LIN {X 0,Y 164.342,Z 168.013,A -85,B 0,C 180,E1 -23364.343,E2 -23364.343} C_VEL
LIN {X 0,Y 164.388,Z 167.994,A -85,B 0,C 180,E1 -23369.135,E2 -23369.135} C_VEL
LIN {X 0,Y 164.405,Z 168.003,A -85,B 0,C 180,E1 -23374.693,E2 -23374.693} C_VEL
LIN {X 0,Y 164.484,Z 167.984,A -85,B 0,C 180,E1 -23380.052,E2 -23380.052} C_VEL
LIN {X 0,Y 164.553,Z 167.979,A -85,B 0,C 180,E1 -23385.152,E2 -23385.152} C_VEL
LIN {X 0,Y 164.809,Z 167.949,A -85,B 0,C 180,E1 -23390.179,E2 -23390.179} C_VEL
LIN {X 0,Y 164.851,Z 167.931,A -85,B 0,C 180,E1 -23392.652,E2 -23392.652} C_VEL
LIN {X 0,Y 165.05,Z 167.922,A -85,B 0,C 180,E1 -23397.56,E2 -23397.56} C_VEL
LIN {X 0,Y 165.296,Z 167.89,A -85,B 0,C 180,E1 -23400.001,E2 -23400.001} C_VEL
LIN {X 0,Y 164.77,Z 167.946,A -85,B 0,C 180,E1 -23404.894,E2 -23404.894} C_VEL
LIN {X 0,Y 164.851,Z 167.948,A -85,B 0,C 180,E1 -23407.349,E2 -23407.349} C_VEL
LIN {X 0,Y 164.754,Z 167.952,A -85,B 0,C 180,E1 -23411.152,E2 -23411.152} C_VEL
LIN {X 0,Y 164.505,Z 167.992,A -85,B 0,C 180,E1 -23417.401,E2 -23417.401} C_VEL
LIN {X 0,Y 164.473,Z 167.988,A -85,B 0,C 180,E1 -23419.99,E2 -23419.99} C_VEL
LIN {X 0,Y 164.387,Z 168.002,A -85,B 0,C 180,E1 -23426.129,E2 -23426.129} C_VEL
LIN {X 0,Y 164.377,Z 168.008,A -85,B 0,C 180,E1 -23431.229,E2 -23431.229} C_VEL
LIN {X 0,Y 164.315,Z 168.017,A -85,B 0,C 180,E1 -23436.785,E2 -23436.785} C_VEL
LIN {X 0,Y 164.307,Z 168.015,A -85,B 0,C 180,E1 -23439.912,E2 -23439.912} C_VEL
LIN {X 0,Y 164.344,Z 168.221,A -85,B 0,C 180,E1 -23444.02,E2 -23444.02} C_VEL
LIN {X 0,Y 165.539,Z 172.969,A -85,B 0,C 180,E1 -23446.861,E2 -23446.861} C_VEL
LIN {X 0,Y 173.075,Z 190.014,A -85,B 0,C 180,E1 -23449.429,E2 -23449.429} C_VEL
LIN {X 0,Y 179.369,Z 206.621,A -85,B 0,C 180,E1 -23451.483,E2 -23451.483} C_VEL
LIN {X 0,Y 181.23,Z 212.268,A -85,B 0,C 180,E1 -23452.102,E2 -23452.102} C_VEL
LIN {X 0,Y 183.794,Z 238.914,A -85,B 0,C 180,E1 -23453.88,E2 -23453.88} C_VEL
LIN {X 0,Y 181.365,Z 282.612,A -85,B 0,C 180,E1 -23455.73,E2 -23455.73} C_VEL
LIN {X 0,Y 180.154,Z 294.602,A -85,B 0,C 180,E1 -23456.562,E2 -23456.562} C_VEL
LIN {X 0,Y 178.065,Z 308.424,A -85,B 0,C 180,E1 -23457.97,E2 -23457.97} C_VEL
LIN {X 0,Y 175.703,Z 320.384,A -85,B 0,C 180,E1 -23459.669,E2 -23459.669} C_VEL
LIN {X 0,Y 173.045,Z 331.876,A -85,B 0,C 180,E1 -23461.827,E2 -23461.827} C_VEL
LIN {X 0,Y 171.732,Z 337.396,A -85,B 0,C 180,E1 -23463.088,E2 -23463.088} C_VEL
LIN {X 0,Y 169.992,Z 341.98,A -85,B 0,C 180,E1 -23464.192,E2 -23464.192} C_VEL
LIN {X 0,Y 165.331,Z 348.901,A -85,B 0,C 180,E1 -23466.027,E2 -23466.027} C_VEL
LIN {X 0,Y 160.682,Z 355.249,A -85,B 0,C 180,E1 -23468.164,E2 -23468.164} C_VEL
LIN {X 0,Y 159.008,Z 358.939,A -85,B 0,C 180,E1 -23469.712,E2 -23469.712} C_VEL
LIN {X 0,Y 157.028,Z 366.916,A -85,B 0,C 180,E1 -23473.756,E2 -23473.756} C_VEL
LIN {X 0,Y 155.91,Z 371.932,A -85,B 0,C 180,E1 -23476.974,E2 -23476.974} C_VEL
LIN {X 0,Y 155.241,Z 376.779,A -85,B 0,C 180,E1 -23480.883,E2 -23480.883} C_VEL
LIN {X 0,Y 155.134,Z 380.873,A -85,B 0,C 180,E1 -23485.323,E2 -23485.323} C_VEL
LIN {X 0,Y 155.163,Z 382.301,A -85,B 0,C 180,E1 -23487.404,E2 -23487.404} C_VEL
LIN {X 0,Y 155.288,Z 383.662,A -85,B 0,C 180,E1 -23490,E2 -23490} C_VEL
LIN {X 0,Y 154.986,Z 384.887,A -85,B 0,C 180,E1 -23493.948,E2 -23493.948} C_VEL
LIN {X 0,Y 154.946,Z 385.166,A -85,B 0,C 180,E1 -23497.821,E2 -23497.821} C_VEL
LIN {X 0,Y 155.286,Z 384.874,A -85,B 0,C 180,E1 -23500.43,E2 -23500.43} C_VEL
LIN {X 0,Y 156.791,Z 383.114,A -85,B 0,C 180,E1 -23505.601,E2 -23505.601} C_VEL
LIN {X 0,Y 159.742,Z 379.828,A -85,B 0,C 180,E1 -23510.607,E2 -23510.607} C_VEL
LIN {X 0,Y 162.745,Z 376.229,A -85,B 0,C 180,E1 -23514.22,E2 -23514.22} C_VEL
LIN {X 0,Y 166.298,Z 371.59,A -85,B 0,C 180,E1 -23517.702,E2 -23517.702} C_VEL
LIN {X 0,Y 171.257,Z 364.691,A -85,B 0,C 180,E1 -23521.549,E2 -23521.549} C_VEL
LIN {X 0,Y 176.322,Z 357.303,A -85,B 0,C 180,E1 -23524.61,E2 -23524.61} C_VEL
LIN {X 0,Y 180.979,Z 349.849,A -85,B 0,C 180,E1 -23527.007,E2 -23527.007} C_VEL
LIN {X 0,Y 185.904,Z 340.918,A -85,B 0,C 180,E1 -23529.288,E2 -23529.288} C_VEL
LIN {X 0,Y 191.245,Z 329.956,A -85,B 0,C 180,E1 -23531.412,E2 -23531.412} C_VEL
LIN {X 0,Y 196.337,Z 317.462,A -85,B 0,C 180,E1 -23533.203,E2 -23533.203} C_VEL
LIN {X 0,Y 200.189,Z 305.943,A -85,B 0,C 180,E1 -23534.422,E2 -23534.422} C_VEL
LIN {X 0,Y 203.607,Z 292.613,A -85,B 0,C 180,E1 -23535.438,E2 -23535.438} C_VEL
LIN {X 0,Y 205.989,Z 279.023,A -85,B 0,C 180,E1 -23536.159,E2 -23536.159} C_VEL
LIN {X 0,Y 209.063,Z 246.653,A -85,B 0,C 180,E1 -23537.336,E2 -23537.336} C_VEL
LIN {X 0,Y 208.859,Z 244.24,A -85,B 0,C 180,E1 -23537.62,E2 -23537.62} C_VEL
LIN {X 0,Y 206.164,Z 236.439,A -85,B 0,C 180,E1 -23539.563,E2 -23539.563} C_VEL
LIN {X 0,Y 202.8,Z 228.202,A -85,B 0,C 180,E1 -23542.218,E2 -23542.218} C_VEL
LIN {X 0,Y 199.99,Z 222.311,A -85,B 0,C 180,E1 -23544.678,E2 -23544.678} C_VEL
LIN {X 0,Y 197.981,Z 218.105,A -85,B 0,C 180,E1 -23546.755,E2 -23546.755} C_VEL
LIN {X 0,Y 195.684,Z 213.557,A -85,B 0,C 180,E1 -23549.537,E2 -23549.537} C_VEL
LIN {X 0,Y 192.783,Z 207.727,A -85,B 0,C 180,E1 -23554.61,E2 -23554.61} C_VEL
LIN {X 0,Y 191.359,Z 205.222,A -85,B 0,C 180,E1 -23559.685,E2 -23559.685} C_VEL
LIN {X 0,Y 191.226,Z 204.943,A -85,B 0,C 180,E1 -23562.901,E2 -23562.901} C_VEL
LIN {X 0,Y 192.564,Z 205.538,A -85,B 0,C 180,E1 -23568.226,E2 -23568.226} C_VEL
LIN {X 0,Y 193.957,Z 208.698,A -85,B 0,C 180,E1 -23571.448,E2 -23571.448} C_VEL
LIN {X 0,Y 196.109,Z 210.925,A -85,B 0,C 180,E1 -23574.391,E2 -23574.391} C_VEL
LIN {X 0,Y 198.35,Z 214.506,A -85,B 0,C 180,E1 -23576.999,E2 -23576.999} C_VEL
LIN {X 0,Y 201.55,Z 219.928,A -85,B 0,C 180,E1 -23580.066,E2 -23580.066} C_VEL
LIN {X 0,Y 204.233,Z 224.357,A -85,B 0,C 180,E1 -23582.176,E2 -23582.176} C_VEL
LIN {X 0,Y 208.74,Z 233.089,A -85,B 0,C 180,E1 -23585.346,E2 -23585.346} C_VEL
LIN {X 0,Y 209.996,Z 235.765,A -85,B 0,C 180,E1 -23586.148,E2 -23586.148} C_VEL
LIN {X 0,Y 206.742,Z 268.852,A -85,B 0,C 180,E1 -23587.35,E2 -23587.35} C_VEL
LIN {X 0,Y 204.486,Z 282.04,A -85,B 0,C 180,E1 -23588.134,E2 -23588.134} C_VEL
LIN {X 0,Y 201.598,Z 294.37,A -85,B 0,C 180,E1 -23589.246,E2 -23589.246} C_VEL
LIN {X 0,Y 197.992,Z 305.927,A -85,B 0,C 180,E1 -23590.642,E2 -23590.642} C_VEL
LIN {X 0,Y 193.662,Z 317.178,A -85,B 0,C 180,E1 -23592.41,E2 -23592.41} C_VEL
LIN {X 0,Y 189.427,Z 326.368,A -85,B 0,C 180,E1 -23594.242,E2 -23594.242} C_VEL
LIN {X 0,Y 184.354,Z 335.943,A -85,B 0,C 180,E1 -23596.717,E2 -23596.717} C_VEL
LIN {X 0,Y 179.038,Z 344.511,A -85,B 0,C 180,E1 -23599.594,E2 -23599.594} C_VEL
LIN {X 0,Y 174.694,Z 350.723,A -85,B 0,C 180,E1 -23602.288,E2 -23602.288} C_VEL
LIN {X 0,Y 170.76,Z 355.834,A -85,B 0,C 180,E1 -23605.116,E2 -23605.116} C_VEL
LIN {X 0,Y 167.247,Z 360.006,A -85,B 0,C 180,E1 -23608.061,E2 -23608.061} C_VEL
LIN {X 0,Y 164.155,Z 363.32,A -85,B 0,C 180,E1 -23611.101,E2 -23611.101} C_VEL
LIN {X 0,Y 161.361,Z 365.976,A -85,B 0,C 180,E1 -23614.486,E2 -23614.486} C_VEL
LIN {X 0,Y 158.921,Z 367.915,A -85,B 0,C 180,E1 -23618.252,E2 -23618.252} C_VEL
LIN {X 0,Y 157.019,Z 368.934,A -85,B 0,C 180,E1 -23622.173,E2 -23622.173} C_VEL
LIN {X 0,Y 155.421,Z 368.889,A -85,B 0,C 180,E1 -23627.29,E2 -23627.29} C_VEL
LIN {X 0,Y 154.873,Z 368.019,A -85,B 0,C 180,E1 -23630.558,E2 -23630.558} C_VEL
LIN {X 0,Y 154.747,Z 365.956,A -85,B 0,C 180,E1 -23634.834,E2 -23634.834} C_VEL
LIN {X 0,Y 155.308,Z 362.591,A -85,B 0,C 180,E1 -23639.292,E2 -23639.292} C_VEL
LIN {X 0,Y 156.23,Z 358.403,A -85,B 0,C 180,E1 -23643.266,E2 -23643.266} C_VEL
LIN {X 0,Y 157.692,Z 352.244,A -85,B 0,C 180,E1 -23647.655,E2 -23647.655} C_VEL
LIN {X 0,Y 159.576,Z 345.482,A -85,B 0,C 180,E1 -23651.379,E2 -23651.379} C_VEL
LIN {X 0,Y 161.81,Z 337.442,A -85,B 0,C 180,E1 -23654.894,E2 -23654.894} C_VEL
LIN {X 0,Y 164.036,Z 329.627,A -85,B 0,C 180,E1 -23657.63,E2 -23657.63} C_VEL
LIN {X 0,Y 166.376,Z 320.404,A -85,B 0,C 180,E1 -23660.272,E2 -23660.272} C_VEL
LIN {X 0,Y 169.033,Z 308.98,A -85,B 0,C 180,E1 -23662.835,E2 -23662.835} C_VEL
LIN {X 0,Y 171.284,Z 298.064,A -85,B 0,C 180,E1 -23664.738,E2 -23664.738} C_VEL
LIN {X 0,Y 173.242,Z 285.976,A -85,B 0,C 180,E1 -23666.366,E2 -23666.366} C_VEL
LIN {X 0,Y 174.897,Z 272.679,A -85,B 0,C 180,E1 -23667.625,E2 -23667.625} C_VEL
LIN {X 0,Y 175.959,Z 259.011,A -85,B 0,C 180,E1 -23668.464,E2 -23668.464} C_VEL
LIN {X 0,Y 178.716,Z 211.992,A -85,B 0,C 180,E1 -23670.441,E2 -23670.441} C_VEL
LIN {X 0,Y 173.825,Z 200.698,A -85,B 0,C 180,E1 -23671.938,E2 -23671.938} C_VEL
LIN {X 0,Y 167.139,Z 185.903,A -85,B 0,C 180,E1 -23674.126,E2 -23674.126} C_VEL
LIN {X 0,Y 158.062,Z 170.127,A -85,B 0,C 180,E1 -23677.148,E2 -23677.148} C_VEL
LIN {X 0,Y 157.784,Z 168.834,A -85,B 0,C 180,E1 -23677.357,E2 -23677.357} C_VEL
LIN {X 0,Y 157.632,Z 168.853,A -85,B 0,C 180,E1 -23681.228,E2 -23681.228} C_VEL
LIN {X 0,Y 157.421,Z 168.875,A -85,B 0,C 180,E1 -23685.537,E2 -23685.537} C_VEL
LIN {X 0,Y 157.356,Z 168.881,A -85,B 0,C 180,E1 -23690.935,E2 -23690.935} C_VEL
LIN {X 0,Y 157.309,Z 168.888,A -85,B 0,C 180,E1 -23696.681,E2 -23696.681} C_VEL
LIN {X 0,Y 157.275,Z 168.894,A -85,B 0,C 180,E1 -23702.427,E2 -23702.427} C_VEL
LIN {X 0,Y 157.267,Z 168.896,A -85,B 0,C 180,E1 -23706.45,E2 -23706.45} C_VEL
LIN {X 0,Y 157.192,Z 168.891,A -85,B 0,C 180,E1 -23712.117,E2 -23712.117} C_VEL
LIN {X 0,Y 157.212,Z 168.895,A -85,B 0,C 180,E1 -23717.89,E2 -23717.89} C_VEL
LIN {X 0,Y 157.282,Z 168.888,A -85,B 0,C 180,E1 -23723.544,E2 -23723.544} C_VEL
LIN {X 0,Y 157.293,Z 168.883,A -85,B 0,C 180,E1 -23728.096,E2 -23728.096} C_VEL
LIN {X 0,Y 157.314,Z 168.881,A -85,B 0,C 180,E1 -23733.465,E2 -23733.465} C_VEL
LIN {X 0,Y 157.391,Z 168.869,A -85,B 0,C 180,E1 -23739.67,E2 -23739.67} C_VEL
LIN {X 0,Y 157.477,Z 168.858,A -85,B 0,C 180,E1 -23744.469,E2 -23744.469} C_VEL
LIN {X 0,Y 157.735,Z 168.831,A -85,B 0,C 180,E1 -23749.734,E2 -23749.734} C_VEL
LIN {X 0,Y 157.809,Z 168.809,A -85,B 0,C 180,E1 -23752.323,E2 -23752.323} C_VEL
LIN {X 0,Y 158.258,Z 168.766,A -85,B 0,C 180,E1 -23760.001,E2 -23760.001} C_VEL
LIN {X 0,Y 157.809,Z 168.825,A -85,B 0,C 180,E1 -23767.679,E2 -23767.679} C_VEL
LIN {X 0,Y 157.684,Z 168.832,A -85,B 0,C 180,E1 -23771.322,E2 -23771.322} C_VEL
LIN {X 0,Y 157.478,Z 168.867,A -85,B 0,C 180,E1 -23775.532,E2 -23775.532} C_VEL
LIN {X 0,Y 157.368,Z 168.874,A -85,B 0,C 180,E1 -23780.934,E2 -23780.934} C_VEL
LIN {X 0,Y 157.31,Z 168.882,A -85,B 0,C 180,E1 -23786.681,E2 -23786.681} C_VEL
LIN {X 0,Y 157.279,Z 168.89,A -85,B 0,C 180,E1 -23792.427,E2 -23792.427} C_VEL
LIN {X 0,Y 157.285,Z 168.894,A -85,B 0,C 180,E1 -23796.458,E2 -23796.458} C_VEL
LIN {X 0,Y 157.266,Z 169.004,A -85,B 0,C 180,E1 -23802.869,E2 -23802.869} C_VEL
LIN {X 0,Y 158.198,Z 172.54,A -85,B 0,C 180,E1 -23805.116,E2 -23805.116} C_VEL
LIN {X 0,Y 165.838,Z 189.387,A -85,B 0,C 180,E1 -23807.891,E2 -23807.891} C_VEL
LIN {X 0,Y 172.101,Z 205.412,A -85,B 0,C 180,E1 -23810.086,E2 -23810.086} C_VEL
LIN {X 0,Y 175.118,Z 214.73,A -85,B 0,C 180,E1 -23811.154,E2 -23811.154} C_VEL
LIN {X 0,Y 177.456,Z 239.19,A -85,B 0,C 180,E1 -23812.848,E2 -23812.848} C_VEL
LIN {X 0,Y 175.301,Z 278.362,A -85,B 0,C 180,E1 -23814.545,E2 -23814.545} C_VEL
LIN {X 0,Y 174.063,Z 291.913,A -85,B 0,C 180,E1 -23815.404,E2 -23815.404} C_VEL
LIN {X 0,Y 172.286,Z 304.181,A -85,B 0,C 180,E1 -23816.585,E2 -23816.585} C_VEL
LIN {X 0,Y 169.943,Z 316.157,A -85,B 0,C 180,E1 -23818.179,E2 -23818.179} C_VEL
LIN {X 0,Y 167.105,Z 328.529,A -85,B 0,C 180,E1 -23820.385,E2 -23820.385} C_VEL
LIN {X 0,Y 164.309,Z 339.453,A -85,B 0,C 180,E1 -23822.97,E2 -23822.97} C_VEL
LIN {X 0,Y 161.528,Z 349.772,A -85,B 0,C 180,E1 -23826.109,E2 -23826.109} C_VEL
LIN {X 0,Y 159.236,Z 358.083,A -85,B 0,C 180,E1 -23829.324,E2 -23829.324} C_VEL
LIN {X 0,Y 159.008,Z 358.939,A -85,B 0,C 180,E1 -23829.712,E2 -23829.712} C_VEL
LIN {X 0,Y 157.448,Z 362.458,A -85,B 0,C 180,E1 -23831.343,E2 -23831.343} C_VEL
LIN {X 0,Y 153.34,Z 367.573,A -85,B 0,C 180,E1 -23834.081,E2 -23834.081} C_VEL
LIN {X 0,Y 149.497,Z 372.037,A -85,B 0,C 180,E1 -23837.112,E2 -23837.112} C_VEL
LIN {X 0,Y 148.399,Z 374.469,A -85,B 0,C 180,E1 -23839.146,E2 -23839.146} C_VEL
LIN {X 0,Y 148.052,Z 378.572,A -85,B 0,C 180,E1 -23843.184,E2 -23843.184} C_VEL
LIN {X 0,Y 148.087,Z 381.615,A -85,B 0,C 180,E1 -23847.28,E2 -23847.28} C_VEL
LIN {X 0,Y 148.222,Z 383.079,A -85,B 0,C 180,E1 -23850,E2 -23850} C_VEL
LIN {X 0,Y 147.917,Z 384.303,A -85,B 0,C 180,E1 -23853.812,E2 -23853.812} C_VEL
LIN {X 0,Y 147.908,Z 384.743,A -85,B 0,C 180,E1 -23858.195,E2 -23858.195} C_VEL
LIN {X 0,Y 148.957,Z 383.928,A -85,B 0,C 180,E1 -23863.645,E2 -23863.645} C_VEL
LIN {X 0,Y 151.349,Z 381.536,A -85,B 0,C 180,E1 -23868.968,E2 -23868.968} C_VEL
LIN {X 0,Y 154.035,Z 378.702,A -85,B 0,C 180,E1 -23872.819,E2 -23872.819} C_VEL
LIN {X 0,Y 158.418,Z 373.749,A -85,B 0,C 180,E1 -23877.466,E2 -23877.466} C_VEL
LIN {X 0,Y 163.646,Z 367.219,A -85,B 0,C 180,E1 -23881.741,E2 -23881.741} C_VEL
LIN {X 0,Y 169.642,Z 359.271,A -85,B 0,C 180,E1 -23885.45,E2 -23885.45} C_VEL
LIN {X 0,Y 174.393,Z 352.266,A -85,B 0,C 180,E1 -23887.92,E2 -23887.92} C_VEL
LIN {X 0,Y 179.444,Z 343.917,A -85,B 0,C 180,E1 -23890.257,E2 -23890.257} C_VEL
LIN {X 0,Y 184.934,Z 333.778,A -85,B 0,C 180,E1 -23892.419,E2 -23892.419} C_VEL
LIN {X 0,Y 190.139,Z 322.487,A -85,B 0,C 180,E1 -23894.24,E2 -23894.24} C_VEL
LIN {X 0,Y 194.335,Z 311.541,A -85,B 0,C 180,E1 -23895.581,E2 -23895.581} C_VEL
LIN {X 0,Y 198.121,Z 299.452,A -85,B 0,C 180,E1 -23896.652,E2 -23896.652} C_VEL
LIN {X 0,Y 201.165,Z 285.726,A -85,B 0,C 180,E1 -23897.548,E2 -23897.548} C_VEL
LIN {X 0,Y 203.122,Z 271.987,A -85,B 0,C 180,E1 -23898.117,E2 -23898.117} C_VEL
LIN {X 0,Y 205.396,Z 248.452,A -85,B 0,C 180,E1 -23898.941,E2 -23898.941} C_VEL
LIN {X 0,Y 203.595,Z 242.578,A -85,B 0,C 180,E1 -23900.393,E2 -23900.393} C_VEL
LIN {X 0,Y 201.126,Z 236.044,A -85,B 0,C 180,E1 -23902.471,E2 -23902.471} C_VEL
LIN {X 0,Y 198.492,Z 229.642,A -85,B 0,C 180,E1 -23904.935,E2 -23904.935} C_VEL
LIN {X 0,Y 195.977,Z 224.178,A -85,B 0,C 180,E1 -23907.666,E2 -23907.666} C_VEL
LIN {X 0,Y 194.072,Z 220.109,A -85,B 0,C 180,E1 -23910.213,E2 -23910.213} C_VEL
LIN {X 0,Y 191.438,Z 214.471,A -85,B 0,C 180,E1 -23915.273,E2 -23915.273} C_VEL
LIN {X 0,Y 190.262,Z 212.115,A -85,B 0,C 180,E1 -23920.228,E2 -23920.228} C_VEL
LIN {X 0,Y 190.501,Z 212.088,A -85,B 0,C 180,E1 -23925.034,E2 -23925.034} C_VEL
LIN {X 0,Y 191.388,Z 212.597,A -85,B 0,C 180,E1 -23927.957,E2 -23927.957} C_VEL
LIN {X 0,Y 192.725,Z 215.646,A -85,B 0,C 180,E1 -23931.174,E2 -23931.174} C_VEL
LIN {X 0,Y 194.592,Z 217.664,A -85,B 0,C 180,E1 -23933.861,E2 -23933.861} C_VEL
LIN {X 0,Y 196.622,Z 221.132,A -85,B 0,C 180,E1 -23936.406,E2 -23936.406} C_VEL
LIN {X 0,Y 199.496,Z 226.202,A -85,B 0,C 180,E1 -23939.31,E2 -23939.31} C_VEL
LIN {X 0,Y 201.913,Z 230.48,A -85,B 0,C 180,E1 -23941.376,E2 -23941.376} C_VEL
LIN {X 0,Y 206.104,Z 239.08,A -85,B 0,C 180,E1 -23944.547,E2 -23944.547} C_VEL
LIN {X 0,Y 203.086,Z 268.927,A -85,B 0,C 180,E1 -23945.642,E2 -23945.642} C_VEL
LIN {X 0,Y 200.697,Z 282.488,A -85,B 0,C 180,E1 -23946.444,E2 -23946.444} C_VEL
LIN {X 0,Y 197.958,Z 293.846,A -85,B 0,C 180,E1 -23947.453,E2 -23947.453} C_VEL
LIN {X 0,Y 194.141,Z 305.774,A -85,B 0,C 180,E1 -23948.852,E2 -23948.852} C_VEL
LIN {X 0,Y 189.396,Z 317.571,A -85,B 0,C 180,E1 -23950.692,E2 -23950.692} C_VEL
LIN {X 0,Y 184.656,Z 327.319,A -85,B 0,C 180,E1 -23952.652,E2 -23952.652} C_VEL
LIN {X 0,Y 179.088,Z 337.139,A -85,B 0,C 180,E1 -23955.273,E2 -23955.273} C_VEL
LIN {X 0,Y 173.827,Z 345.138,A -85,B 0,C 180,E1 -23958.014,E2 -23958.014} C_VEL
LIN {X 0,Y 168.094,Z 352.817,A -85,B 0,C 180,E1 -23961.524,E2 -23961.524} C_VEL
LIN {X 0,Y 163.075,Z 358.645,A -85,B 0,C 180,E1 -23965.173,E2 -23965.173} C_VEL
LIN {X 0,Y 158.587,Z 363.239,A -85,B 0,C 180,E1 -23969.174,E2 -23969.174} C_VEL
LIN {X 0,Y 155.258,Z 366.199,A -85,B 0,C 180,E1 -23972.901,E2 -23972.901} C_VEL
LIN {X 0,Y 151.797,Z 368.685,A -85,B 0,C 180,E1 -23978.087,E2 -23978.087} C_VEL
LIN {X 0,Y 150.147,Z 369.393,A -85,B 0,C 180,E1 -23981.504,E2 -23981.504} C_VEL
LIN {X 0,Y 148.858,Z 369.45,A -85,B 0,C 180,E1 -23985.087,E2 -23985.087} C_VEL
LIN {X 0,Y 147.914,Z 368.582,A -85,B 0,C 180,E1 -23989.483,E2 -23989.483} C_VEL
LIN {X 0,Y 147.641,Z 366.602,A -85,B 0,C 180,E1 -23994.02,E2 -23994.02} C_VEL
LIN {X 0,Y 148.083,Z 363.365,A -85,B 0,C 180,E1 -23998.679,E2 -23998.679} C_VEL
LIN {X 0,Y 149.188,Z 358.566,A -85,B 0,C 180,E1 -24003.515,E2 -24003.515} C_VEL
LIN {X 0,Y 150.705,Z 352.34,A -85,B 0,C 180,E1 -24008.095,E2 -24008.095} C_VEL
LIN {X 0,Y 152.593,Z 345.772,A -85,B 0,C 180,E1 -24011.849,E2 -24011.849} C_VEL
LIN {X 0,Y 154.951,Z 337.61,A -85,B 0,C 180,E1 -24015.555,E2 -24015.555} C_VEL
LIN {X 0,Y 157.618,Z 328.514,A -85,B 0,C 180,E1 -24018.796,E2 -24018.796} C_VEL
LIN {X 0,Y 160.414,Z 317.771,A -85,B 0,C 180,E1 -24021.814,E2 -24021.814} C_VEL
LIN {X 0,Y 163.036,Z 306.867,A -85,B 0,C 180,E1 -24024.203,E2 -24024.203} C_VEL
LIN {X 0,Y 165.389,Z 295.046,A -85,B 0,C 180,E1 -24026.193,E2 -24026.193} C_VEL
LIN {X 0,Y 167.313,Z 282.616,A -85,B 0,C 180,E1 -24027.769,E2 -24027.769} C_VEL
LIN {X 0,Y 168.859,Z 269.265,A -85,B 0,C 180,E1 -24028.949,E2 -24028.949} C_VEL
LIN {X 0,Y 170.055,Z 252.532,A -85,B 0,C 180,E1 -24029.814,E2 -24029.814} C_VEL
LIN {X 0,Y 172.487,Z 213.896,A -85,B 0,C 180,E1 -24031.472,E2 -24031.472} C_VEL
LIN {X 0,Y 162.052,Z 190.204,A -85,B 0,C 180,E1 -24034.976,E2 -24034.976} C_VEL
LIN {X 0,Y 152.338,Z 173.468,A -85,B 0,C 180,E1 -24038.411,E2 -24038.411} C_VEL
LIN {X 0,Y 150.851,Z 170.754,A -85,B 0,C 180,E1 -24038.99,E2 -24038.99} C_VEL
LIN {X 0,Y 150.641,Z 169.724,A -85,B 0,C 180,E1 -24039.144,E2 -24039.144} C_VEL
LIN {X 0,Y 150.415,Z 169.75,A -85,B 0,C 180,E1 -24043.51,E2 -24043.51} C_VEL
LIN {X 0,Y 150.316,Z 169.761,A -85,B 0,C 180,E1 -24049.104,E2 -24049.104} C_VEL
LIN {X 0,Y 150.258,Z 169.766,A -85,B 0,C 180,E1 -24051.974,E2 -24051.974} C_VEL
LIN {X 0,Y 150.219,Z 169.769,A -85,B 0,C 180,E1 -24057.895,E2 -24057.895} C_VEL
LIN {X 0,Y 150.215,Z 169.774,A -85,B 0,C 180,E1 -24062.633,E2 -24062.633} C_VEL
LIN {X 0,Y 150.172,Z 169.778,A -85,B 0,C 180,E1 -24067.473,E2 -24067.473} C_VEL
LIN {X 0,Y 150.135,Z 169.768,A -85,B 0,C 180,E1 -24071.499,E2 -24071.499} C_VEL
LIN {X 0,Y 150.125,Z 169.783,A -85,B 0,C 180,E1 -24075.396,E2 -24075.396} C_VEL
LIN {X 0,Y 150.155,Z 169.767,A -85,B 0,C 180,E1 -24079.06,E2 -24079.06} C_VEL
LIN {X 0,Y 150.215,Z 169.765,A -85,B 0,C 180,E1 -24082.69,E2 -24082.69} C_VEL
LIN {X 0,Y 150.217,Z 169.768,A -85,B 0,C 180,E1 -24087.367,E2 -24087.367} C_VEL
LIN {X 0,Y 150.24,Z 169.757,A -85,B 0,C 180,E1 -24092.721,E2 -24092.721} C_VEL
LIN {X 0,Y 150.349,Z 169.749,A -85,B 0,C 180,E1 -24099.21,E2 -24099.21} C_VEL
LIN {X 0,Y 150.381,Z 169.734,A -85,B 0,C 180,E1 -24103.716,E2 -24103.716} C_VEL
LIN {X 0,Y 150.658,Z 169.715,A -85,B 0,C 180,E1 -24109.246,E2 -24109.246} C_VEL
LIN {X 0,Y 150.745,Z 169.691,A -85,B 0,C 180,E1 -24111.961,E2 -24111.961} C_VEL
LIN {X 0,Y 151.218,Z 169.643,A -85,B 0,C 180,E1 -24120.001,E2 -24120.001} C_VEL
LIN {X 0,Y 150.745,Z 169.705,A -85,B 0,C 180,E1 -24128.041,E2 -24128.041} C_VEL
LIN {X 0,Y 150.615,Z 169.711,A -85,B 0,C 180,E1 -24131.508,E2 -24131.508} C_VEL
LIN {X 0,Y 150.383,Z 169.752,A -85,B 0,C 180,E1 -24136.285,E2 -24136.285} C_VEL
LIN {X 0,Y 150.35,Z 169.747,A -85,B 0,C 180,E1 -24140.791,E2 -24140.791} C_VEL
LIN {X 0,Y 150.242,Z 169.763,A -85,B 0,C 180,E1 -24147.28,E2 -24147.28} C_VEL
LIN {X 0,Y 150.22,Z 169.769,A -85,B 0,C 180,E1 -24152.635,E2 -24152.635} C_VEL
LIN {X 0,Y 150.213,Z 169.773,A -85,B 0,C 180,E1 -24157.462,E2 -24157.462} C_VEL
LIN {X 0,Y 150.204,Z 169.887,A -85,B 0,C 180,E1 -24161.687,E2 -24161.687} C_VEL
LIN {X 0,Y 150.835,Z 172.283,A -85,B 0,C 180,E1 -24163.198,E2 -24163.198} C_VEL
LIN {X 0,Y 157.459,Z 186.301,A -85,B 0,C 180,E1 -24165.803,E2 -24165.803} C_VEL
LIN {X 0,Y 163.398,Z 200.467,A -85,B 0,C 180,E1 -24168.014,E2 -24168.014} C_VEL
LIN {X 0,Y 168.966,Z 216.152,A -85,B 0,C 180,E1 -24170.072,E2 -24170.072} C_VEL
LIN {X 0,Y 171.184,Z 240.306,A -85,B 0,C 180,E1 -24171.822,E2 -24171.822} C_VEL
LIN {X 0,Y 168.623,Z 281.802,A -85,B 0,C 180,E1 -24173.684,E2 -24173.684} C_VEL
LIN {X 0,Y 167.244,Z 294.301,A -85,B 0,C 180,E1 -24174.611,E2 -24174.611} C_VEL
LIN {X 0,Y 165.121,Z 307.439,A -85,B 0,C 180,E1 -24176.039,E2 -24176.039} C_VEL
LIN {X 0,Y 162.798,Z 318.664,A -85,B 0,C 180,E1 -24177.708,E2 -24177.708} C_VEL
LIN {X 0,Y 159.921,Z 330.32,A -85,B 0,C 180,E1 -24180.007,E2 -24180.007} C_VEL
LIN {X 0,Y 157.075,Z 340.86,A -85,B 0,C 180,E1 -24182.702,E2 -24182.702} C_VEL
LIN {X 0,Y 154.379,Z 350.369,A -85,B 0,C 180,E1 -24185.813,E2 -24185.813} C_VEL
LIN {X 0,Y 152.021,Z 358.692,A -85,B 0,C 180,E1 -24189.28,E2 -24189.28} C_VEL
LIN {X 0,Y 150.195,Z 365.773,A -85,B 0,C 180,E1 -24192.995,E2 -24192.995} C_VEL
LIN {X 0,Y 148.641,Z 372.754,A -85,B 0,C 180,E1 -24197.715,E2 -24197.715} C_VEL
LIN {X 0,Y 148.399,Z 374.469,A -85,B 0,C 180,E1 -24199.146,E2 -24199.146} C_VEL
LIN {X 0,Y 147.514,Z 376.713,A -85,B 0,C 180,E1 -24201.246,E2 -24201.246} C_VEL
LIN {X 0,Y 145.911,Z 378.574,A -85,B 0,C 180,E1 -24203.358,E2 -24203.358} C_VEL
LIN {X 0,Y 142.31,Z 381.408,A -85,B 0,C 180,E1 -24207.763,E2 -24207.763} C_VEL
LIN {X 0,Y 141.036,Z 382.773,A -85,B 0,C 180,E1 -24210.907,E2 -24210.907} C_VEL
LIN {X 0,Y 140.847,Z 383.68,A -85,B 0,C 180,E1 -24213.65,E2 -24213.65} C_VEL
LIN {X 0,Y 140.865,Z 384.318,A -85,B 0,C 180,E1 -24218.608,E2 -24218.608} C_VEL
LIN {X 0,Y 142.025,Z 383.642,A -85,B 0,C 180,E1 -24224.325,E2 -24224.325} C_VEL
LIN {X 0,Y 143.091,Z 382.726,A -85,B 0,C 180,E1 -24227.139,E2 -24227.139} C_VEL
LIN {X 0,Y 146.456,Z 379.707,A -85,B 0,C 180,E1 -24232.575,E2 -24232.575} C_VEL
LIN {X 0,Y 149.867,Z 376.379,A -85,B 0,C 180,E1 -24236.455,E2 -24236.455} C_VEL
LIN {X 0,Y 153.856,Z 372.044,A -85,B 0,C 180,E1 -24240.163,E2 -24240.163} C_VEL
LIN {X 0,Y 159.381,Z 365.568,A -85,B 0,C 180,E1 -24244.209,E2 -24244.209} C_VEL
LIN {X 0,Y 164.923,Z 358.61,A -85,B 0,C 180,E1 -24247.39,E2 -24247.39} C_VEL
LIN {X 0,Y 169.958,Z 351.596,A -85,B 0,C 180,E1 -24249.862,E2 -24249.862} C_VEL
LIN {X 0,Y 175.263,Z 343.247,A -85,B 0,C 180,E1 -24252.196,E2 -24252.196} C_VEL
LIN {X 0,Y 180.985,Z 333.041,A -85,B 0,C 180,E1 -24254.344,E2 -24254.344} C_VEL
LIN {X 0,Y 186.416,Z 321.673,A -85,B 0,C 180,E1 -24256.139,E2 -24256.139} C_VEL
LIN {X 0,Y 190.811,Z 310.613,A -85,B 0,C 180,E1 -24257.446,E2 -24257.446} C_VEL
LIN {X 0,Y 194.689,Z 298.332,A -85,B 0,C 180,E1 -24258.507,E2 -24258.507} C_VEL
LIN {X 0,Y 197.802,Z 284.7,A -85,B 0,C 180,E1 -24259.363,E2 -24259.363} C_VEL
LIN {X 0,Y 199.819,Z 270.614,A -85,B 0,C 180,E1 -24259.932,E2 -24259.932} C_VEL
LIN {X 0,Y 201.784,Z 251.146,A -85,B 0,C 180,E1 -24260.623,E2 -24260.623} C_VEL
LIN {X 0,Y 199.755,Z 244.632,A -85,B 0,C 180,E1 -24262.461,E2 -24262.461} C_VEL
LIN {X 0,Y 197.201,Z 237.874,A -85,B 0,C 180,E1 -24264.931,E2 -24264.931} C_VEL
LIN {X 0,Y 195.171,Z 232.892,A -85,B 0,C 180,E1 -24267.195,E2 -24267.195} C_VEL
LIN {X 0,Y 193.748,Z 229.638,A -85,B 0,C 180,E1 -24268.991,E2 -24268.991} C_VEL
LIN {X 0,Y 192.417,Z 226.51,A -85,B 0,C 180,E1 -24271.014,E2 -24271.014} C_VEL
LIN {X 0,Y 190.21,Z 221.333,A -85,B 0,C 180,E1 -24275.704,E2 -24275.704} C_VEL
LIN {X 0,Y 189.204,Z 219.082,A -85,B 0,C 180,E1 -24280.469,E2 -24280.469} C_VEL
LIN {X 0,Y 189.655,Z 219.194,A -85,B 0,C 180,E1 -24285.883,E2 -24285.883} C_VEL
LIN {X 0,Y 190.187,Z 219.531,A -85,B 0,C 180,E1 -24287.578,E2 -24287.578} C_VEL
LIN {X 0,Y 191.617,Z 222.73,A -85,B 0,C 180,E1 -24291.105,E2 -24291.105} C_VEL
LIN {X 0,Y 193.139,Z 224.471,A -85,B 0,C 180,E1 -24293.388,E2 -24293.388} C_VEL
LIN {X 0,Y 194.834,Z 227.55,A -85,B 0,C 180,E1 -24295.68,E2 -24295.68} C_VEL
LIN {X 0,Y 197.562,Z 232.625,A -85,B 0,C 180,E1 -24298.624,E2 -24298.624} C_VEL
LIN {X 0,Y 199.631,Z 236.619,A -85,B 0,C 180,E1 -24300.56,E2 -24300.56} C_VEL
LIN {X 0,Y 202.504,Z 242.708,A -85,B 0,C 180,E1 -24302.906,E2 -24302.906} C_VEL
LIN {X 0,Y 199.492,Z 270.355,A -85,B 0,C 180,E1 -24303.935,E2 -24303.935} C_VEL
LIN {X 0,Y 197.048,Z 283.31,A -85,B 0,C 180,E1 -24304.704,E2 -24304.704} C_VEL
LIN {X 0,Y 193.811,Z 295.764,A -85,B 0,C 180,E1 -24305.836,E2 -24305.836} C_VEL
LIN {X 0,Y 189.595,Z 307.97,A -85,B 0,C 180,E1 -24307.321,E2 -24307.321} C_VEL
LIN {X 0,Y 185.015,Z 318.68,A -85,B 0,C 180,E1 -24309.021,E2 -24309.021} C_VEL
LIN {X 0,Y 179.836,Z 328.696,A -85,B 0,C 180,E1 -24311.074,E2 -24311.074} C_VEL
LIN {X 0,Y 174.396,Z 337.782,A -85,B 0,C 180,E1 -24313.541,E2 -24313.541} C_VEL
LIN {X 0,Y 168.556,Z 346.129,A -85,B 0,C 180,E1 -24316.467,E2 -24316.467} C_VEL
LIN {X 0,Y 163.749,Z 352.156,A -85,B 0,C 180,E1 -24319.228,E2 -24319.228} C_VEL
LIN {X 0,Y 158.13,Z 358.438,A -85,B 0,C 180,E1 -24323.044,E2 -24323.044} C_VEL
LIN {X 0,Y 152.977,Z 363.407,A -85,B 0,C 180,E1 -24327.349,E2 -24327.349} C_VEL
LIN {X 0,Y 148.8,Z 366.827,A -85,B 0,C 180,E1 -24331.772,E2 -24331.772} C_VEL
LIN {X 0,Y 146.293,Z 368.533,A -85,B 0,C 180,E1 -24335.246,E2 -24335.246} C_VEL
LIN {X 0,Y 143.915,Z 369.673,A -85,B 0,C 180,E1 -24339.408,E2 -24339.408} C_VEL
LIN {X 0,Y 142.104,Z 369.897,A -85,B 0,C 180,E1 -24343.819,E2 -24343.819} C_VEL
LIN {X 0,Y 141,Z 369.118,A -85,B 0,C 180,E1 -24348.387,E2 -24348.387} C_VEL
LIN {X 0,Y 140.583,Z 366.262,A -85,B 0,C 180,E1 -24354.907,E2 -24354.907} C_VEL
LIN {X 0,Y 141.227,Z 362.32,A -85,B 0,C 180,E1 -24360.157,E2 -24360.157} C_VEL
LIN {X 0,Y 142.532,Z 356.968,A -85,B 0,C 180,E1 -24365.221,E2 -24365.221} C_VEL
LIN {X 0,Y 144.026,Z 351.392,A -85,B 0,C 180,E1 -24369.237,E2 -24369.237} C_VEL
LIN {X 0,Y 146.149,Z 344.355,A -85,B 0,C 180,E1 -24373.23,E2 -24373.23} C_VEL
LIN {X 0,Y 148.721,Z 335.845,A -85,B 0,C 180,E1 -24377.022,E2 -24377.022} C_VEL
LIN {X 0,Y 151.46,Z 326.498,A -85,B 0,C 180,E1 -24380.317,E2 -24380.317} C_VEL
LIN {X 0,Y 154.364,Z 315.801,A -85,B 0,C 180,E1 -24383.272,E2 -24383.272} C_VEL
LIN {X 0,Y 157.25,Z 303.682,A -85,B 0,C 180,E1 -24385.835,E2 -24385.835} C_VEL
LIN {X 0,Y 159.631,Z 291.822,A -85,B 0,C 180,E1 -24387.741,E2 -24387.741} C_VEL
LIN {X 0,Y 161.528,Z 278.723,A -85,B 0,C 180,E1 -24389.287,E2 -24389.287} C_VEL
LIN {X 0,Y 163.026,Z 264.858,A -85,B 0,C 180,E1 -24390.374,E2 -24390.374} C_VEL
LIN {X 0,Y 166.145,Z 215.482,A -85,B 0,C 180,E1 -24392.634,E2 -24392.634} C_VEL
LIN {X 0,Y 156.64,Z 193.899,A -85,B 0,C 180,E1 -24396,E2 -24396} C_VEL
LIN {X 0,Y 147.172,Z 177.573,A -85,B 0,C 180,E1 -24399.545,E2 -24399.545} C_VEL
LIN {X 0,Y 145.365,Z 174.506,A -85,B 0,C 180,E1 -24400.277,E2 -24400.277} C_VEL
LIN {X 0,Y 143.846,Z 171.904,A -85,B 0,C 180,E1 -24400.914,E2 -24400.914} C_VEL
LIN {X 0,Y 143.557,Z 170.606,A -85,B 0,C 180,E1 -24401.119,E2 -24401.119} C_VEL
LIN {X 0,Y 143.268,Z 170.638,A -85,B 0,C 180,E1 -24407.117,E2 -24407.117} C_VEL
LIN {X 0,Y 143.267,Z 170.636,A -85,B 0,C 180,E1 -24411.244,E2 -24411.244} C_VEL
LIN {X 0,Y 143.188,Z 170.645,A -85,B 0,C 180,E1 -24417.936,E2 -24417.936} C_VEL
LIN {X 0,Y 143.143,Z 170.654,A -85,B 0,C 180,E1 -24423.42,E2 -24423.42} C_VEL
LIN {X 0,Y 143.054,Z 170.654,A -85,B 0,C 180,E1 -24429.692,E2 -24429.692} C_VEL
LIN {X 0,Y 143.033,Z 170.663,A -85,B 0,C 180,E1 -24433.464,E2 -24433.464} C_VEL
LIN {X 0,Y 143.066,Z 170.659,A -85,B 0,C 180,E1 -24437.464,E2 -24437.464} C_VEL
LIN {X 0,Y 143.105,Z 170.644,A -85,B 0,C 180,E1 -24441.792,E2 -24441.792} C_VEL
LIN {X 0,Y 143.184,Z 170.644,A -85,B 0,C 180,E1 -24447.323,E2 -24447.323} C_VEL
LIN {X 0,Y 143.187,Z 170.628,A -85,B 0,C 180,E1 -24452.065,E2 -24452.065} C_VEL
LIN {X 0,Y 143.274,Z 170.633,A -85,B 0,C 180,E1 -24458.748,E2 -24458.748} C_VEL
LIN {X 0,Y 143.315,Z 170.609,A -85,B 0,C 180,E1 -24462.889,E2 -24462.889} C_VEL
LIN {X 0,Y 143.594,Z 170.596,A -85,B 0,C 180,E1 -24468.711,E2 -24468.711} C_VEL
LIN {X 0,Y 143.665,Z 170.574,A -85,B 0,C 180,E1 -24471.562,E2 -24471.562} C_VEL
LIN {X 0,Y 144.177,Z 170.52,A -85,B 0,C 180,E1 -24480.001,E2 -24480.001} C_VEL
LIN {X 0,Y 143.665,Z 170.587,A -85,B 0,C 180,E1 -24488.44,E2 -24488.44} C_VEL
LIN {X 0,Y 143.549,Z 170.59,A -85,B 0,C 180,E1 -24491.713,E2 -24491.713} C_VEL
LIN {X 0,Y 143.317,Z 170.632,A -85,B 0,C 180,E1 -24497.112,E2 -24497.112} C_VEL
LIN {X 0,Y 143.276,Z 170.63,A -85,B 0,C 180,E1 -24501.253,E2 -24501.253} C_VEL
LIN {X 0,Y 143.189,Z 170.645,A -85,B 0,C 180,E1 -24507.936,E2 -24507.936} C_VEL
LIN {X 0,Y 143.17,Z 170.651,A -85,B 0,C 180,E1 -24513.436,E2 -24513.436} C_VEL
LIN {X 0,Y 143.084,Z 170.658,A -85,B 0,C 180,E1 -24519.683,E2 -24519.683} C_VEL
LIN {X 0,Y 143.115,Z 170.728,A -85,B 0,C 180,E1 -24520.362,E2 -24520.362} C_VEL
LIN {X 0,Y 143.323,Z 171.597,A -85,B 0,C 180,E1 -24520.985,E2 -24520.985} C_VEL
LIN {X 0,Y 149.993,Z 185.192,A -85,B 0,C 180,E1 -24523.836,E2 -24523.836} C_VEL
LIN {X 0,Y 155.64,Z 198.19,A -85,B 0,C 180,E1 -24526.117,E2 -24526.117} C_VEL
LIN {X 0,Y 161.8,Z 214.767,A -85,B 0,C 180,E1 -24528.514,E2 -24528.514} C_VEL
LIN {X 0,Y 163.101,Z 219.422,A -85,B 0,C 180,E1 -24529.063,E2 -24529.063} C_VEL
LIN {X 0,Y 164.898,Z 241.934,A -85,B 0,C 180,E1 -24530.735,E2 -24530.735} C_VEL
LIN {X 0,Y 162.26,Z 282.19,A -85,B 0,C 180,E1 -24532.61,E2 -24532.61} C_VEL
LIN {X 0,Y 160.819,Z 294.378,A -85,B 0,C 180,E1 -24533.554,E2 -24533.554} C_VEL
LIN {X 0,Y 158.641,Z 307.413,A -85,B 0,C 180,E1 -24535.03,E2 -24535.03} C_VEL
LIN {X 0,Y 156.037,Z 319.328,A -85,B 0,C 180,E1 -24536.899,E2 -24536.899} C_VEL
LIN {X 0,Y 153.069,Z 330.788,A -85,B 0,C 180,E1 -24539.283,E2 -24539.283} C_VEL
LIN {X 0,Y 150.119,Z 341.179,A -85,B 0,C 180,E1 -24542.085,E2 -24542.085} C_VEL
LIN {X 0,Y 147.35,Z 350.526,A -85,B 0,C 180,E1 -24545.333,E2 -24545.333} C_VEL
LIN {X 0,Y 144.743,Z 359.61,A -85,B 0,C 180,E1 -24549.389,E2 -24549.389} C_VEL
LIN {X 0,Y 142.749,Z 366.878,A -85,B 0,C 180,E1 -24553.555,E2 -24553.555} C_VEL
LIN {X 0,Y 141.665,Z 371.759,A -85,B 0,C 180,E1 -24557.1,E2 -24557.1} C_VEL
LIN {X 0,Y 141.031,Z 376.466,A -85,B 0,C 180,E1 -24561.402,E2 -24561.402} C_VEL
LIN {X 0,Y 140.991,Z 379.863,A -85,B 0,C 180,E1 -24565.526,E2 -24565.526} C_VEL
LIN {X 0,Y 141.157,Z 382.44,A -85,B 0,C 180,E1 -24570,E2 -24570} C_VEL
LIN {X 0,Y 141.036,Z 382.773,A -85,B 0,C 180,E1 -24570.907,E2 -24570.907} C_VEL
LIN {X 0,Y 140.155,Z 383.532,A -85,B 0,C 180,E1 -24573.268,E2 -24573.268} C_VEL
LIN {X 0,Y 137.236,Z 384.004,A -85,B 0,C 180,E1 -24577.181,E2 -24577.181} C_VEL
LIN {X 0,Y 135.121,Z 383.969,A -85,B 0,C 180,E1 -24580.428,E2 -24580.428} C_VEL
LIN {X 0,Y 134.582,Z 383.716,A -85,B 0,C 180,E1 -24582.945,E2 -24582.945} C_VEL
LIN {X 0,Y 134.723,Z 383.537,A -85,B 0,C 180,E1 -24583.786,E2 -24583.786} C_VEL
LIN {X 0,Y 136.292,Z 382.509,A -85,B 0,C 180,E1 -24588.022,E2 -24588.022} C_VEL
LIN {X 0,Y 137.948,Z 381.299,A -85,B 0,C 180,E1 -24590.893,E2 -24590.893} C_VEL
LIN {X 0,Y 141.025,Z 378.719,A -85,B 0,C 180,E1 -24595.062,E2 -24595.062} C_VEL
LIN {X 0,Y 145.276,Z 374.758,A -85,B 0,C 180,E1 -24599.449,E2 -24599.449} C_VEL
LIN {X 0,Y 150.933,Z 368.895,A -85,B 0,C 180,E1 -24603.97,E2 -24603.97} C_VEL
LIN {X 0,Y 157.366,Z 361.693,A -85,B 0,C 180,E1 -24607.884,E2 -24607.884} C_VEL
LIN {X 0,Y 163.523,Z 353.943,A -85,B 0,C 180,E1 -24610.951,E2 -24610.951} C_VEL
LIN {X 0,Y 170.12,Z 344.356,A -85,B 0,C 180,E1 -24613.786,E2 -24613.786} C_VEL
LIN {X 0,Y 176.067,Z 334.542,A -85,B 0,C 180,E1 -24615.93,E2 -24615.93} C_VEL
LIN {X 0,Y 181.656,Z 323.713,A -85,B 0,C 180,E1 -24617.724,E2 -24617.724} C_VEL
LIN {X 0,Y 186.141,Z 313.297,A -85,B 0,C 180,E1 -24619.036,E2 -24619.036} C_VEL
LIN {X 0,Y 190.509,Z 300.942,A -85,B 0,C 180,E1 -24620.155,E2 -24620.155} C_VEL
LIN {X 0,Y 193.85,Z 288.095,A -85,B 0,C 180,E1 -24621.035,E2 -24621.035} C_VEL
LIN {X 0,Y 196.281,Z 273.857,A -85,B 0,C 180,E1 -24621.658,E2 -24621.658} C_VEL
LIN {X 0,Y 198.426,Z 254.07,A -85,B 0,C 180,E1 -24622.339,E2 -24622.339} C_VEL
LIN {X 0,Y 196.175,Z 247.064,A -85,B 0,C 180,E1 -24624.612,E2 -24624.612} C_VEL
LIN {X 0,Y 193.946,Z 240.871,A -85,B 0,C 180,E1 -24627.18,E2 -24627.18} C_VEL
LIN {X 0,Y 192.271,Z 236.539,A -85,B 0,C 180,E1 -24629.438,E2 -24629.438} C_VEL
LIN {X 0,Y 190.797,Z 232.921,A -85,B 0,C 180,E1 -24631.831,E2 -24631.831} C_VEL
LIN {X 0,Y 189.006,Z 228.205,A -85,B 0,C 180,E1 -24636.11,E2 -24636.11} C_VEL
LIN {X 0,Y 188.171,Z 226.169,A -85,B 0,C 180,E1 -24640.358,E2 -24640.358} C_VEL
LIN {X 0,Y 188.391,Z 226.122,A -85,B 0,C 180,E1 -24644.862,E2 -24644.862} C_VEL
LIN {X 0,Y 189.006,Z 226.514,A -85,B 0,C 180,E1 -24647.239,E2 -24647.239} C_VEL
LIN {X 0,Y 190.371,Z 229.632,A -85,B 0,C 180,E1 -24650.776,E2 -24650.776} C_VEL
LIN {X 0,Y 191.749,Z 231.385,A -85,B 0,C 180,E1 -24652.992,E2 -24652.992} C_VEL
LIN {X 0,Y 193.174,Z 234.176,A -85,B 0,C 180,E1 -24655.04,E2 -24655.04} C_VEL
LIN {X 0,Y 196.348,Z 240.266,A -85,B 0,C 180,E1 -24658.615,E2 -24658.615} C_VEL
LIN {X 0,Y 199.067,Z 246.387,A -85,B 0,C 180,E1 -24661.203,E2 -24661.203} C_VEL
LIN {X 0,Y 196.263,Z 270.935,A -85,B 0,C 180,E1 -24662.116,E2 -24662.116} C_VEL
LIN {X 0,Y 193.797,Z 283.569,A -85,B 0,C 180,E1 -24662.855,E2 -24662.855} C_VEL
LIN {X 0,Y 190.634,Z 295.417,A -85,B 0,C 180,E1 -24663.896,E2 -24663.896} C_VEL
LIN {X 0,Y 186.181,Z 307.895,A -85,B 0,C 180,E1 -24665.377,E2 -24665.377} C_VEL
LIN {X 0,Y 181.255,Z 318.931,A -85,B 0,C 180,E1 -24667.105,E2 -24667.105} C_VEL
LIN {X 0,Y 175.67,Z 329.225,A -85,B 0,C 180,E1 -24669.208,E2 -24669.208} C_VEL
LIN {X 0,Y 169.285,Z 339.286,A -85,B 0,C 180,E1 -24671.98,E2 -24671.98} C_VEL
LIN {X 0,Y 163.096,Z 347.545,A -85,B 0,C 180,E1 -24674.983,E2 -24674.983} C_VEL
LIN {X 0,Y 157.343,Z 354.172,A -85,B 0,C 180,E1 -24678.219,E2 -24678.219} C_VEL
LIN {X 0,Y 151.649,Z 359.92,A -85,B 0,C 180,E1 -24682.048,E2 -24682.048} C_VEL
LIN {X 0,Y 145.772,Z 365.012,A -85,B 0,C 180,E1 -24687,E2 -24687} C_VEL
LIN {X 0,Y 141.129,Z 368.267,A -85,B 0,C 180,E1 -24692.16,E2 -24692.16} C_VEL
LIN {X 0,Y 137.504,Z 370.052,A -85,B 0,C 180,E1 -24697.83,E2 -24697.83} C_VEL
LIN {X 0,Y 135.13,Z 370.266,A -85,B 0,C 180,E1 -24703.271,E2 -24703.271} C_VEL
LIN {X 0,Y 134.102,Z 369.638,A -85,B 0,C 180,E1 -24707.198,E2 -24707.198} C_VEL
LIN {X 0,Y 133.478,Z 367.857,A -85,B 0,C 180,E1 -24712.165,E2 -24712.165} C_VEL
LIN {X 0,Y 133.688,Z 364.86,A -85,B 0,C 180,E1 -24717.258,E2 -24717.258} C_VEL
LIN {X 0,Y 134.651,Z 360.37,A -85,B 0,C 180,E1 -24722.535,E2 -24722.535} C_VEL
LIN {X 0,Y 135.91,Z 355.419,A -85,B 0,C 180,E1 -24726.9,E2 -24726.9} C_VEL
LIN {X 0,Y 137.878,Z 348.83,A -85,B 0,C 180,E1 -24731.423,E2 -24731.423} C_VEL
LIN {X 0,Y 140.266,Z 341.239,A -85,B 0,C 180,E1 -24735.492,E2 -24735.492} C_VEL
LIN {X 0,Y 143.068,Z 332.278,A -85,B 0,C 180,E1 -24739.253,E2 -24739.253} C_VEL
LIN {X 0,Y 146.201,Z 321.632,A -85,B 0,C 180,E1 -24742.751,E2 -24742.751} C_VEL
LIN {X 0,Y 149.252,Z 310.198,A -85,B 0,C 180,E1 -24745.612,E2 -24745.612} C_VEL
LIN {X 0,Y 152.124,Z 297.605,A -85,B 0,C 180,E1 -24748.014,E2 -24748.014} C_VEL
LIN {X 0,Y 154.174,Z 285.972,A -85,B 0,C 180,E1 -24749.674,E2 -24749.674} C_VEL
LIN {X 0,Y 156.054,Z 272.065,A -85,B 0,C 180,E1 -24751.068,E2 -24751.068} C_VEL
LIN {X 0,Y 157.171,Z 259.22,A -85,B 0,C 180,E1 -24751.878,E2 -24751.878} C_VEL
LIN {X 0,Y 159.994,Z 217.448,A -85,B 0,C 180,E1 -24753.791,E2 -24753.791} C_VEL
LIN {X 0,Y 151.427,Z 197.867,A -85,B 0,C 180,E1 -24757.041,E2 -24757.041} C_VEL
LIN {X 0,Y 142.37,Z 182.011,A -85,B 0,C 180,E1 -24760.627,E2 -24760.627} C_VEL
LIN {X 0,Y 138.644,Z 175.868,A -85,B 0,C 180,E1 -24762.258,E2 -24762.258} C_VEL
LIN {X 0,Y 136.908,Z 173.557,A -85,B 0,C 180,E1 -24763.013,E2 -24763.013} C_VEL
LIN {X 0,Y 136.312,Z 171.506,A -85,B 0,C 180,E1 -24763.38,E2 -24763.38} C_VEL
LIN {X 0,Y 136.187,Z 171.518,A -85,B 0,C 180,E1 -24768.037,E2 -24768.037} C_VEL
LIN {X 0,Y 136.189,Z 171.518,A -85,B 0,C 180,E1 -24771.74,E2 -24771.74} C_VEL
LIN {X 0,Y 136.098,Z 171.53,A -85,B 0,C 180,E1 -24778.615,E2 -24778.615} C_VEL
LIN {X 0,Y 136.042,Z 171.536,A -85,B 0,C 180,E1 -24784.629,E2 -24784.629} C_VEL
LIN {X 0,Y 136.026,Z 171.533,A -85,B 0,C 180,E1 -24789.196,E2 -24789.196} C_VEL
LIN {X 0,Y 135.978,Z 171.542,A -85,B 0,C 180,E1 -24793.65,E2 -24793.65} C_VEL
LIN {X 0,Y 136.03,Z 171.532,A -85,B 0,C 180,E1 -24797.807,E2 -24797.807} C_VEL
LIN {X 0,Y 136.054,Z 171.521,A -85,B 0,C 180,E1 -24801.694,E2 -24801.694} C_VEL
LIN {X 0,Y 136.089,Z 171.532,A -85,B 0,C 180,E1 -24805.718,E2 -24805.718} C_VEL
LIN {X 0,Y 136.143,Z 171.507,A -85,B 0,C 180,E1 -24812.316,E2 -24812.316} C_VEL
LIN {X 0,Y 136.241,Z 171.508,A -85,B 0,C 180,E1 -24818.833,E2 -24818.833} C_VEL
LIN {X 0,Y 136.283,Z 171.499,A -85,B 0,C 180,E1 -24825.058,E2 -24825.058} C_VEL
LIN {X 0,Y 136.497,Z 171.48,A -85,B 0,C 180,E1 -24828.115,E2 -24828.115} C_VEL
LIN {X 0,Y 136.592,Z 171.456,A -85,B 0,C 180,E1 -24831.121,E2 -24831.121} C_VEL
LIN {X 0,Y 137.134,Z 171.397,A -85,B 0,C 180,E1 -24840.001,E2 -24840.001} C_VEL
LIN {X 0,Y 136.592,Z 171.468,A -85,B 0,C 180,E1 -24848.88,E2 -24848.88} C_VEL
LIN {X 0,Y 136.492,Z 171.467,A -85,B 0,C 180,E1 -24851.955,E2 -24851.955} C_VEL
LIN {X 0,Y 136.252,Z 171.51,A -85,B 0,C 180,E1 -24858.029,E2 -24858.029} C_VEL
LIN {X 0,Y 136.197,Z 171.514,A -85,B 0,C 180,E1 -24861.747,E2 -24861.747} C_VEL
LIN {X 0,Y 136.1,Z 171.531,A -85,B 0,C 180,E1 -24868.616,E2 -24868.616} C_VEL
LIN {X 0,Y 136.08,Z 171.536,A -85,B 0,C 180,E1 -24874.619,E2 -24874.619} C_VEL
LIN {X 0,Y 136.068,Z 171.59,A -85,B 0,C 180,E1 -24878.627,E2 -24878.627} C_VEL
LIN {X 0,Y 136.963,Z 174.202,A -85,B 0,C 180,E1 -24879.139,E2 -24879.139} C_VEL
LIN {X 0,Y 138.838,Z 176.882,A -85,B 0,C 180,E1 -24879.967,E2 -24879.967} C_VEL
LIN {X 0,Y 144.718,Z 188.742,A -85,B 0,C 180,E1 -24882.619,E2 -24882.619} C_VEL
LIN {X 0,Y 150.766,Z 202.966,A -85,B 0,C 180,E1 -24885.22,E2 -24885.22} C_VEL
LIN {X 0,Y 156.567,Z 219.291,A -85,B 0,C 180,E1 -24887.653,E2 -24887.653} C_VEL
LIN {X 0,Y 157.14,Z 222.297,A -85,B 0,C 180,E1 -24887.965,E2 -24887.965} C_VEL
LIN {X 0,Y 158.718,Z 242.362,A -85,B 0,C 180,E1 -24889.516,E2 -24889.516} C_VEL
LIN {X 0,Y 156.006,Z 281.862,A -85,B 0,C 180,E1 -24891.417,E2 -24891.417} C_VEL
LIN {X 0,Y 154.602,Z 293.569,A -85,B 0,C 180,E1 -24892.349,E2 -24892.349} C_VEL
LIN {X 0,Y 152.219,Z 307.231,A -85,B 0,C 180,E1 -24893.937,E2 -24893.937} C_VEL
LIN {X 0,Y 149.705,Z 318.283,A -85,B 0,C 180,E1 -24895.712,E2 -24895.712} C_VEL
LIN {X 0,Y 146.629,Z 329.854,A -85,B 0,C 180,E1 -24898.181,E2 -24898.181} C_VEL
LIN {X 0,Y 143.552,Z 340.33,A -85,B 0,C 180,E1 -24901.089,E2 -24901.089} C_VEL
LIN {X 0,Y 140.632,Z 349.814,A -85,B 0,C 180,E1 -24904.485,E2 -24904.485} C_VEL
LIN {X 0,Y 138.058,Z 358.217,A -85,B 0,C 180,E1 -24908.342,E2 -24908.342} C_VEL
LIN {X 0,Y 135.954,Z 365.672,A -85,B 0,C 180,E1 -24912.708,E2 -24912.708} C_VEL
LIN {X 0,Y 134.721,Z 370.696,A -85,B 0,C 180,E1 -24916.423,E2 -24916.423} C_VEL
LIN {X 0,Y 134.002,Z 375.548,A -85,B 0,C 180,E1 -24920.947,E2 -24920.947} C_VEL
LIN {X 0,Y 133.915,Z 379.347,A -85,B 0,C 180,E1 -24925.673,E2 -24925.673} C_VEL
LIN {X 0,Y 134.092,Z 381.784,A -85,B 0,C 180,E1 -24930,E2 -24930} C_VEL
LIN {X 0,Y 133.788,Z 383.066,A -85,B 0,C 180,E1 -24933.536,E2 -24933.536} C_VEL
LIN {X 0,Y 133.825,Z 383.893,A -85,B 0,C 180,E1 -24939.064,E2 -24939.064} C_VEL
LIN {X 0,Y 134.723,Z 383.537,A -85,B 0,C 180,E1 -24943.786,E2 -24943.786} C_VEL
LIN {X 0,Y 134.901,Z 383.058,A -85,B 0,C 180,E1 -24946.287,E2 -24946.287} C_VEL
LIN {X 0,Y 134.004,Z 381.663,A -85,B 0,C 180,E1 -24950.457,E2 -24950.457} C_VEL
LIN {X 0,Y 133.865,Z 379.743,A -85,B 0,C 180,E1 -24954.609,E2 -24954.609} C_VEL
LIN {X 0,Y 135.193,Z 378.21,A -85,B 0,C 180,E1 -24956.974,E2 -24956.974} C_VEL
LIN {X 0,Y 140.151,Z 373.996,A -85,B 0,C 180,E1 -24961.769,E2 -24961.769} C_VEL
LIN {X 0,Y 145.115,Z 369.277,A -85,B 0,C 180,E1 -24965.532,E2 -24965.532} C_VEL
LIN {X 0,Y 151.85,Z 362.252,A -85,B 0,C 180,E1 -24969.522,E2 -24969.522} C_VEL
LIN {X 0,Y 158.278,Z 354.747,A -85,B 0,C 180,E1 -24972.62,E2 -24972.62} C_VEL
LIN {X 0,Y 165.138,Z 345.545,A -85,B 0,C 180,E1 -24975.467,E2 -24975.467} C_VEL
LIN {X 0,Y 171.909,Z 335.045,A -85,B 0,C 180,E1 -24977.815,E2 -24977.815} C_VEL
LIN {X 0,Y 177.706,Z 324.464,A -85,B 0,C 180,E1 -24979.579,E2 -24979.579} C_VEL
LIN {X 0,Y 182.325,Z 314.338,A -85,B 0,C 180,E1 -24980.872,E2 -24980.872} C_VEL
LIN {X 0,Y 187.158,Z 301.309,A -85,B 0,C 180,E1 -24982.052,E2 -24982.052} C_VEL
LIN {X 0,Y 190.733,Z 288.254,A -85,B 0,C 180,E1 -24982.934,E2 -24982.934} C_VEL
LIN {X 0,Y 193.231,Z 274.582,A -85,B 0,C 180,E1 -24983.525,E2 -24983.525} C_VEL
LIN {X 0,Y 195.223,Z 257.21,A -85,B 0,C 180,E1 -24984.131,E2 -24984.131} C_VEL
LIN {X 0,Y 193.277,Z 250.68,A -85,B 0,C 180,E1 -24986.447,E2 -24986.447} C_VEL
LIN {X 0,Y 191.002,Z 243.941,A -85,B 0,C 180,E1 -24989.584,E2 -24989.584} C_VEL
LIN {X 0,Y 189.308,Z 239.498,A -85,B 0,C 180,E1 -24992.49,E2 -24992.49} C_VEL
LIN {X 0,Y 187.732,Z 234.909,A -85,B 0,C 180,E1 -24996.77,E2 -24996.77} C_VEL
LIN {X 0,Y 187.14,Z 233.236,A -85,B 0,C 180,E1 -25000.245,E2 -25000.245} C_VEL
LIN {X 0,Y 187.054,Z 232.98,A -85,B 0,C 180,E1 -25002.507,E2 -25002.507} C_VEL
LIN {X 0,Y 187.819,Z 233.471,A -85,B 0,C 180,E1 -25006.849,E2 -25006.849} C_VEL
LIN {X 0,Y 189.409,Z 236.952,A -85,B 0,C 180,E1 -25011,E2 -25011} C_VEL
LIN {X 0,Y 190.264,Z 238.063,A -85,B 0,C 180,E1 -25012.418,E2 -25012.418} C_VEL
LIN {X 0,Y 191.55,Z 240.788,A -85,B 0,C 180,E1 -25014.4,E2 -25014.4} C_VEL
LIN {X 0,Y 194.305,Z 246.436,A -85,B 0,C 180,E1 -25017.77,E2 -25017.77} C_VEL
LIN {X 0,Y 195.847,Z 250.177,A -85,B 0,C 180,E1 -25019.415,E2 -25019.415} C_VEL
LIN {X 0,Y 193.18,Z 272.117,A -85,B 0,C 180,E1 -25020.259,E2 -25020.259} C_VEL
LIN {X 0,Y 190.427,Z 285.306,A -85,B 0,C 180,E1 -25021.047,E2 -25021.047} C_VEL
LIN {X 0,Y 186.849,Z 297.556,A -85,B 0,C 180,E1 -25022.155,E2 -25022.155} C_VEL
LIN {X 0,Y 182.505,Z 309.026,A -85,B 0,C 180,E1 -25023.523,E2 -25023.523} C_VEL
LIN {X 0,Y 177.621,Z 319.489,A -85,B 0,C 180,E1 -25025.154,E2 -25025.154} C_VEL
LIN {X 0,Y 171.664,Z 329.96,A -85,B 0,C 180,E1 -25027.277,E2 -25027.277} C_VEL
LIN {X 0,Y 165.542,Z 339.129,A -85,B 0,C 180,E1 -25029.777,E2 -25029.777} C_VEL
LIN {X 0,Y 158.645,Z 347.898,A -85,B 0,C 180,E1 -25032.943,E2 -25032.943} C_VEL
LIN {X 0,Y 151.725,Z 355.352,A -85,B 0,C 180,E1 -25036.672,E2 -25036.672} C_VEL
LIN {X 0,Y 145.59,Z 361.086,A -85,B 0,C 180,E1 -25040.694,E2 -25040.694} C_VEL
LIN {X 0,Y 139.94,Z 365.553,A -85,B 0,C 180,E1 -25045.314,E2 -25045.314} C_VEL
LIN {X 0,Y 136.427,Z 367.898,A -85,B 0,C 180,E1 -25048.867,E2 -25048.867} C_VEL
LIN {X 0,Y 133.443,Z 369.502,A -85,B 0,C 180,E1 -25052.578,E2 -25052.578} C_VEL
LIN {X 0,Y 131.01,Z 370.472,A -85,B 0,C 180,E1 -25056.422,E2 -25056.422} C_VEL
LIN {X 0,Y 128.862,Z 370.765,A -85,B 0,C 180,E1 -25060.879,E2 -25060.879} C_VEL
LIN {X 0,Y 127.247,Z 370.127,A -85,B 0,C 180,E1 -25065.889,E2 -25065.889} C_VEL
LIN {X 0,Y 126.375,Z 367.876,A -85,B 0,C 180,E1 -25072.285,E2 -25072.285} C_VEL
LIN {X 0,Y 126.716,Z 364.272,A -85,B 0,C 180,E1 -25078.294,E2 -25078.294} C_VEL
LIN {X 0,Y 127.871,Z 359.362,A -85,B 0,C 180,E1 -25083.916,E2 -25083.916} C_VEL
LIN {X 0,Y 129.369,Z 353.876,A -85,B 0,C 180,E1 -25088.623,E2 -25088.623} C_VEL
LIN {X 0,Y 131.804,Z 346.186,A -85,B 0,C 180,E1 -25093.695,E2 -25093.695} C_VEL
LIN {X 0,Y 134.557,Z 337.807,A -85,B 0,C 180,E1 -25097.941,E2 -25097.941} C_VEL
LIN {X 0,Y 137.895,Z 327.528,A -85,B 0,C 180,E1 -25101.943,E2 -25101.943} C_VEL
LIN {X 0,Y 141.058,Z 316.782,A -85,B 0,C 180,E1 -25105.179,E2 -25105.179} C_VEL
LIN {X 0,Y 144.145,Z 304.87,A -85,B 0,C 180,E1 -25107.905,E2 -25107.905} C_VEL
LIN {X 0,Y 146.788,Z 292.771,A -85,B 0,C 180,E1 -25110,E2 -25110} C_VEL
LIN {X 0,Y 148.926,Z 279.335,A -85,B 0,C 180,E1 -25111.69,E2 -25111.69} C_VEL
LIN {X 0,Y 150.501,Z 265.833,A -85,B 0,C 180,E1 -25112.818,E2 -25112.818} C_VEL
LIN {X 0,Y 153.822,Z 219.394,A -85,B 0,C 180,E1 -25115.059,E2 -25115.059} C_VEL
LIN {X 0,Y 146.191,Z 201.699,A -85,B 0,C 180,E1 -25118.15,E2 -25118.15} C_VEL
LIN {X 0,Y 137.47,Z 186.236,A -85,B 0,C 180,E1 -25121.85,E2 -25121.85} C_VEL
LIN {X 0,Y 133.953,Z 180.608,A -85,B 0,C 180,E1 -25123.472,E2 -25123.472} C_VEL
LIN {X 0,Y 131.931,Z 177.336,A -85,B 0,C 180,E1 -25124.449,E2 -25124.449} C_VEL
LIN {X 0,Y 129.661,Z 174.298,A -85,B 0,C 180,E1 -25125.545,E2 -25125.545} C_VEL
LIN {X 0,Y 129.13,Z 172.4,A -85,B 0,C 180,E1 -25125.994,E2 -25125.994} C_VEL
LIN {X 0,Y 129.106,Z 172.402,A -85,B 0,C 180,E1 -25132.399,E2 -25132.399} C_VEL
LIN {X 0,Y 129.026,Z 172.412,A -85,B 0,C 180,E1 -25135.833,E2 -25135.833} C_VEL
LIN {X 0,Y 129.016,Z 172.413,A -85,B 0,C 180,E1 -25139.358,E2 -25139.358} C_VEL
LIN {X 0,Y 128.958,Z 172.419,A -85,B 0,C 180,E1 -25145.168,E2 -25145.168} C_VEL
LIN {X 0,Y 128.923,Z 172.408,A -85,B 0,C 180,E1 -25150.856,E2 -25150.856} C_VEL
LIN {X 0,Y 128.917,Z 172.425,A -85,B 0,C 180,E1 -25155.129,E2 -25155.129} C_VEL
LIN {X 0,Y 128.956,Z 172.401,A -85,B 0,C 180,E1 -25159.728,E2 -25159.728} C_VEL
LIN {X 0,Y 128.991,Z 172.415,A -85,B 0,C 180,E1 -25164.811,E2 -25164.811} C_VEL
LIN {X 0,Y 129.016,Z 172.388,A -85,B 0,C 180,E1 -25170.643,E2 -25170.643} C_VEL
LIN {X 0,Y 129.026,Z 172.406,A -85,B 0,C 180,E1 -25174.167,E2 -25174.167} C_VEL
LIN {X 0,Y 129.106,Z 172.4,A -85,B 0,C 180,E1 -25177.729,E2 -25177.729} C_VEL
LIN {X 0,Y 129.158,Z 172.373,A -85,B 0,C 180,E1 -25180.945,E2 -25180.945} C_VEL
LIN {X 0,Y 129.416,Z 172.363,A -85,B 0,C 180,E1 -25187.821,E2 -25187.821} C_VEL
LIN {X 0,Y 129.518,Z 172.34,A -85,B 0,C 180,E1 -25190.632,E2 -25190.632} C_VEL
LIN {X 0,Y 130.089,Z 172.275,A -85,B 0,C 180,E1 -25200.001,E2 -25200.001} C_VEL
LIN {X 0,Y 129.518,Z 172.348,A -85,B 0,C 180,E1 -25209.369,E2 -25209.369} C_VEL
LIN {X 0,Y 129.394,Z 172.35,A -85,B 0,C 180,E1 -25212.549,E2 -25212.549} C_VEL
LIN {X 0,Y 129.159,Z 172.387,A -85,B 0,C 180,E1 -25219.056,E2 -25219.056} C_VEL
LIN {X 0,Y 129.108,Z 172.4,A -85,B 0,C 180,E1 -25222.399,E2 -25222.399} C_VEL
LIN {X 0,Y 129.037,Z 172.414,A -85,B 0,C 180,E1 -25229.374,E2 -25229.374} C_VEL
LIN {X 0,Y 128.976,Z 172.42,A -85,B 0,C 180,E1 -25235.784,E2 -25235.784} C_VEL
LIN {X 0,Y 128.981,Z 172.434,A -85,B 0,C 180,E1 -25236.107,E2 -25236.107} C_VEL
LIN {X 0,Y 129.845,Z 175.03,A -85,B 0,C 180,E1 -25236.662,E2 -25236.662} C_VEL
LIN {X 0,Y 131.765,Z 177.62,A -85,B 0,C 180,E1 -25237.594,E2 -25237.594} C_VEL
LIN {X 0,Y 134.745,Z 182.594,A -85,B 0,C 180,E1 -25239.04,E2 -25239.04} C_VEL
LIN {X 0,Y 139.693,Z 192.862,A -85,B 0,C 180,E1 -25241.435,E2 -25241.435} C_VEL
LIN {X 0,Y 144.682,Z 204.686,A -85,B 0,C 180,E1 -25243.722,E2 -25243.722} C_VEL
LIN {X 0,Y 150.483,Z 220.957,A -85,B 0,C 180,E1 -25246.33,E2 -25246.33} C_VEL
LIN {X 0,Y 151.227,Z 224.813,A -85,B 0,C 180,E1 -25246.761,E2 -25246.761} C_VEL
LIN {X 0,Y 152.555,Z 242.705,A -85,B 0,C 180,E1 -25248.214,E2 -25248.214} C_VEL
LIN {X 0,Y 149.782,Z 281.604,A -85,B 0,C 180,E1 -25250.151,E2 -25250.151} C_VEL
LIN {X 0,Y 148.181,Z 293.974,A -85,B 0,C 180,E1 -25251.175,E2 -25251.175} C_VEL
LIN {X 0,Y 145.854,Z 306.907,A -85,B 0,C 180,E1 -25252.748,E2 -25252.748} C_VEL
LIN {X 0,Y 143.048,Z 318.733,A -85,B 0,C 180,E1 -25254.74,E2 -25254.74} C_VEL
LIN {X 0,Y 139.856,Z 330.15,A -85,B 0,C 180,E1 -25257.303,E2 -25257.303} C_VEL
LIN {X 0,Y 136.676,Z 340.509,A -85,B 0,C 180,E1 -25260.335,E2 -25260.335} C_VEL
LIN {X 0,Y 133.72,Z 349.701,A -85,B 0,C 180,E1 -25263.821,E2 -25263.821} C_VEL
LIN {X 0,Y 131.024,Z 358.198,A -85,B 0,C 180,E1 -25267.947,E2 -25267.947} C_VEL
LIN {X 0,Y 128.839,Z 365.583,A -85,B 0,C 180,E1 -25272.541,E2 -25272.541} C_VEL
LIN {X 0,Y 127.451,Z 371.464,A -85,B 0,C 180,E1 -25277.257,E2 -25277.257} C_VEL
LIN {X 0,Y 126.849,Z 376.047,A -85,B 0,C 180,E1 -25282.038,E2 -25282.038} C_VEL
LIN {X 0,Y 126.858,Z 379.471,A -85,B 0,C 180,E1 -25286.824,E2 -25286.824} C_VEL
LIN {X 0,Y 127.028,Z 381.127,A -85,B 0,C 180,E1 -25290,E2 -25290} C_VEL
LIN {X 0,Y 126.742,Z 382.398,A -85,B 0,C 180,E1 -25293.5,E2 -25293.5} C_VEL
LIN {X 0,Y 126.807,Z 383.455,A -85,B 0,C 180,E1 -25299.571,E2 -25299.571} C_VEL
LIN {X 0,Y 128.234,Z 383.036,A -85,B 0,C 180,E1 -25305.904,E2 -25305.904} C_VEL
LIN {X 0,Y 131.319,Z 381.14,A -85,B 0,C 180,E1 -25312.001,E2 -25312.001} C_VEL
LIN {X 0,Y 135.193,Z 378.21,A -85,B 0,C 180,E1 -25316.974,E2 -25316.974} C_VEL
LIN {X 0,Y 136.726,Z 376.566,A -85,B 0,C 180,E1 -25319.278,E2 -25319.278} C_VEL
LIN {X 0,Y 137.944,Z 373.501,A -85,B 0,C 180,E1 -25323.187,E2 -25323.187} C_VEL
LIN {X 0,Y 139.72,Z 369.814,A -85,B 0,C 180,E1 -25326.908,E2 -25326.908} C_VEL
LIN {X 0,Y 142.031,Z 367.189,A -85,B 0,C 180,E1 -25328.836,E2 -25328.836} C_VEL
LIN {X 0,Y 148.662,Z 360.626,A -85,B 0,C 180,E1 -25332.351,E2 -25332.351} C_VEL
LIN {X 0,Y 154.364,Z 354.251,A -85,B 0,C 180,E1 -25334.885,E2 -25334.885} C_VEL
LIN {X 0,Y 161.552,Z 345.023,A -85,B 0,C 180,E1 -25337.693,E2 -25337.693} C_VEL
LIN {X 0,Y 168.587,Z 334.502,A -85,B 0,C 180,E1 -25339.996,E2 -25339.996} C_VEL
LIN {X 0,Y 174.603,Z 323.91,A -85,B 0,C 180,E1 -25341.711,E2 -25341.711} C_VEL
LIN {X 0,Y 179.431,Z 313.783,A -85,B 0,C 180,E1 -25342.944,E2 -25342.944} C_VEL
LIN {X 0,Y 183.966,Z 302.067,A -85,B 0,C 180,E1 -25343.998,E2 -25343.998} C_VEL
LIN {X 0,Y 187.941,Z 288.378,A -85,B 0,C 180,E1 -25344.907,E2 -25344.907} C_VEL
LIN {X 0,Y 190.583,Z 274.813,A -85,B 0,C 180,E1 -25345.489,E2 -25345.489} C_VEL
LIN {X 0,Y 192.28,Z 260.471,A -85,B 0,C 180,E1 -25346.005,E2 -25346.005} C_VEL
LIN {X 0,Y 190.467,Z 254.214,A -85,B 0,C 180,E1 -25348.482,E2 -25348.482} C_VEL
LIN {X 0,Y 188.859,Z 249.042,A -85,B 0,C 180,E1 -25351.18,E2 -25351.18} C_VEL
LIN {X 0,Y 187.762,Z 245.782,A -85,B 0,C 180,E1 -25353.415,E2 -25353.415} C_VEL
LIN {X 0,Y 186.543,Z 241.795,A -85,B 0,C 180,E1 -25357.192,E2 -25357.192} C_VEL
LIN {X 0,Y 186.049,Z 240.169,A -85,B 0,C 180,E1 -25360.798,E2 -25360.798} C_VEL
LIN {X 0,Y 186.612,Z 240.285,A -85,B 0,C 180,E1 -25366.202,E2 -25366.202} C_VEL
LIN {X 0,Y 188.571,Z 244.337,A -85,B 0,C 180,E1 -25371.426,E2 -25371.426} C_VEL
LIN {X 0,Y 189.834,Z 247.055,A -85,B 0,C 180,E1 -25373.553,E2 -25373.553} C_VEL
LIN {X 0,Y 192.379,Z 252.804,A -85,B 0,C 180,E1 -25376.998,E2 -25376.998} C_VEL
LIN {X 0,Y 192.891,Z 254.087,A -85,B 0,C 180,E1 -25377.595,E2 -25377.595} C_VEL
LIN {X 0,Y 190.43,Z 273.114,A -85,B 0,C 180,E1 -25378.33,E2 -25378.33} C_VEL
LIN {X 0,Y 187.887,Z 284.856,A -85,B 0,C 180,E1 -25379.002,E2 -25379.002} C_VEL
LIN {X 0,Y 184.471,Z 296.527,A -85,B 0,C 180,E1 -25380,E2 -25380} C_VEL
LIN {X 0,Y 180.206,Z 307.651,A -85,B 0,C 180,E1 -25381.256,E2 -25381.256} C_VEL
LIN {X 0,Y 175.035,Z 318.483,A -85,B 0,C 180,E1 -25382.846,E2 -25382.846} C_VEL
LIN {X 0,Y 168.596,Z 329.591,A -85,B 0,C 180,E1 -25384.999,E2 -25384.999} C_VEL
LIN {X 0,Y 162.126,Z 338.955,A -85,B 0,C 180,E1 -25387.472,E2 -25387.472} C_VEL
LIN {X 0,Y 155.218,Z 347.433,A -85,B 0,C 180,E1 -25390.434,E2 -25390.434} C_VEL
LIN {X 0,Y 148.697,Z 354.286,A -85,B 0,C 180,E1 -25393.669,E2 -25393.669} C_VEL
LIN {X 0,Y 142.72,Z 359.719,A -85,B 0,C 180,E1 -25397.185,E2 -25397.185} C_VEL
LIN {X 0,Y 136.235,Z 364.715,A -85,B 0,C 180,E1 -25401.788,E2 -25401.788} C_VEL
LIN {X 0,Y 132.211,Z 367.387,A -85,B 0,C 180,E1 -25405.355,E2 -25405.355} C_VEL
LIN {X 0,Y 128.349,Z 369.493,A -85,B 0,C 180,E1 -25409.525,E2 -25409.525} C_VEL
LIN {X 0,Y 124.978,Z 370.797,A -85,B 0,C 180,E1 -25414.217,E2 -25414.217} C_VEL
LIN {X 0,Y 122.364,Z 371.179,A -85,B 0,C 180,E1 -25419.181,E2 -25419.181} C_VEL
LIN {X 0,Y 120.217,Z 370.394,A -85,B 0,C 180,E1 -25425.451,E2 -25425.451} C_VEL
LIN {X 0,Y 119.47,Z 368.999,A -85,B 0,C 180,E1 -25429.883,E2 -25429.883} C_VEL
LIN {X 0,Y 119.328,Z 366.227,A -85,B 0,C 180,E1 -25435.542,E2 -25435.542} C_VEL
LIN {X 0,Y 120.107,Z 362.051,A -85,B 0,C 180,E1 -25441.367,E2 -25441.367} C_VEL
LIN {X 0,Y 121.349,Z 357.532,A -85,B 0,C 180,E1 -25446.083,E2 -25446.083} C_VEL
LIN {X 0,Y 123.516,Z 350.383,A -85,B 0,C 180,E1 -25451.763,E2 -25451.763} C_VEL
LIN {X 0,Y 126.054,Z 342.969,A -85,B 0,C 180,E1 -25456.293,E2 -25456.293} C_VEL
LIN {X 0,Y 129.14,Z 333.888,A -85,B 0,C 180,E1 -25460.604,E2 -25460.604} C_VEL
LIN {X 0,Y 132.571,Z 323.434,A -85,B 0,C 180,E1 -25464.416,E2 -25464.416} C_VEL
LIN {X 0,Y 135.744,Z 312.822,A -85,B 0,C 180,E1 -25467.404,E2 -25467.404} C_VEL
LIN {X 0,Y 138.813,Z 300.688,A -85,B 0,C 180,E1 -25470,E2 -25470} C_VEL
LIN {X 0,Y 141.222,Z 288.942,A -85,B 0,C 180,E1 -25471.899,E2 -25471.899} C_VEL
LIN {X 0,Y 143.228,Z 276.073,A -85,B 0,C 180,E1 -25473.399,E2 -25473.399} C_VEL
LIN {X 0,Y 144.702,Z 262.255,A -85,B 0,C 180,E1 -25474.42,E2 -25474.42} C_VEL
LIN {X 0,Y 147.645,Z 221.219,A -85,B 0,C 180,E1 -25476.455,E2 -25476.455} C_VEL
LIN {X 0,Y 140.868,Z 205.259,A -85,B 0,C 180,E1 -25479.388,E2 -25479.388} C_VEL
LIN {X 0,Y 131.794,Z 188.948,A -85,B 0,C 180,E1 -25483.553,E2 -25483.553} C_VEL
LIN {X 0,Y 126.677,Z 181.266,A -85,B 0,C 180,E1 -25486.105,E2 -25486.105} C_VEL
LIN {X 0,Y 124.28,Z 177.555,A -85,B 0,C 180,E1 -25487.421,E2 -25487.421} C_VEL
LIN {X 0,Y 122.685,Z 175.416,A -85,B 0,C 180,E1 -25488.303,E2 -25488.303} C_VEL
LIN {X 0,Y 122.074,Z 173.277,A -85,B 0,C 180,E1 -25488.788,E2 -25488.788} C_VEL
LIN {X 0,Y 121.981,Z 173.287,A -85,B 0,C 180,E1 -25493.785,E2 -25493.785} C_VEL
LIN {X 0,Y 121.926,Z 173.296,A -85,B 0,C 180,E1 -25500.161,E2 -25500.161} C_VEL
LIN {X 0,Y 121.882,Z 173.302,A -85,B 0,C 180,E1 -25506.171,E2 -25506.171} C_VEL
LIN {X 0,Y 121.863,Z 173.287,A -85,B 0,C 180,E1 -25511.434,E2 -25511.434} C_VEL
LIN {X 0,Y 121.883,Z 173.288,A -85,B 0,C 180,E1 -25518.556,E2 -25518.556} C_VEL
LIN {X 0,Y 121.944,Z 173.293,A -85,B 0,C 180,E1 -25524.808,E2 -25524.808} C_VEL
LIN {X 0,Y 121.929,Z 173.272,A -85,B 0,C 180,E1 -25529.837,E2 -25529.837} C_VEL
LIN {X 0,Y 121.982,Z 173.29,A -85,B 0,C 180,E1 -25536.216,E2 -25536.216} C_VEL
LIN {X 0,Y 122.048,Z 173.268,A -85,B 0,C 180,E1 -25539.788,E2 -25539.788} C_VEL
LIN {X 0,Y 122.264,Z 173.252,A -85,B 0,C 180,E1 -25546.708,E2 -25546.708} C_VEL
LIN {X 0,Y 122.447,Z 173.225,A -85,B 0,C 180,E1 -25550.086,E2 -25550.086} C_VEL
LIN {X 0,Y 122.606,Z 173.203,A -85,B 0,C 180,E1 -25556.715,E2 -25556.715} C_VEL
LIN {X 0,Y 123.043,Z 173.152,A -85,B 0,C 180,E1 -25560.001,E2 -25560.001} C_VEL
LIN {X 0,Y 122.446,Z 173.225,A -85,B 0,C 180,E1 -25566.592,E2 -25566.592} C_VEL
LIN {X 0,Y 122.447,Z 173.227,A -85,B 0,C 180,E1 -25569.916,E2 -25569.916} C_VEL
LIN {X 0,Y 122.264,Z 173.239,A -85,B 0,C 180,E1 -25573.294,E2 -25573.294} C_VEL
LIN {X 0,Y 122.048,Z 173.269,A -85,B 0,C 180,E1 -25580.213,E2 -25580.213} C_VEL
LIN {X 0,Y 121.983,Z 173.291,A -85,B 0,C 180,E1 -25583.786,E2 -25583.786} C_VEL
LIN {X 0,Y 121.943,Z 173.297,A -85,B 0,C 180,E1 -25590.174,E2 -25590.174} C_VEL
LIN {X 0,Y 121.946,Z 173.292,A -85,B 0,C 180,E1 -25593.197,E2 -25593.197} C_VEL
LIN {X 0,Y 123.118,Z 176.417,A -85,B 0,C 180,E1 -25594.066,E2 -25594.066} C_VEL
LIN {X 0,Y 124.821,Z 178.548,A -85,B 0,C 180,E1 -25594.975,E2 -25594.975} C_VEL
LIN {X 0,Y 127.007,Z 181.943,A -85,B 0,C 180,E1 -25596.156,E2 -25596.156} C_VEL
LIN {X 0,Y 130.706,Z 188.178,A -85,B 0,C 180,E1 -25598.074,E2 -25598.074} C_VEL
LIN {X 0,Y 136.47,Z 200.993,A -85,B 0,C 180,E1 -25601.042,E2 -25601.042} C_VEL
LIN {X 0,Y 141.866,Z 214.919,A -85,B 0,C 180,E1 -25603.667,E2 -25603.667} C_VEL
LIN {X 0,Y 145.24,Z 225.422,A -85,B 0,C 180,E1 -25605.294,E2 -25605.294} C_VEL
LIN {X 0,Y 146.462,Z 243.405,A -85,B 0,C 180,E1 -25606.824,E2 -25606.824} C_VEL
LIN {X 0,Y 143.635,Z 281.341,A -85,B 0,C 180,E1 -25608.775,E2 -25608.775} C_VEL
LIN {X 0,Y 141.979,Z 293.674,A -85,B 0,C 180,E1 -25609.831,E2 -25609.831} C_VEL
LIN {X 0,Y 139.55,Z 306.579,A -85,B 0,C 180,E1 -25611.448,E2 -25611.448} C_VEL
LIN {X 0,Y 136.411,Z 319.17,A -85,B 0,C 180,E1 -25613.666,E2 -25613.666} C_VEL
LIN {X 0,Y 133.137,Z 330.452,A -85,B 0,C 180,E1 -25616.339,E2 -25616.339} C_VEL
LIN {X 0,Y 129.835,Z 340.661,A -85,B 0,C 180,E1 -25619.505,E2 -25619.505} C_VEL
LIN {X 0,Y 126.83,Z 349.558,A -85,B 0,C 180,E1 -25623.076,E2 -25623.076} C_VEL
LIN {X 0,Y 123.976,Z 358.153,A -85,B 0,C 180,E1 -25627.502,E2 -25627.502} C_VEL
LIN {X 0,Y 121.72,Z 365.465,A -85,B 0,C 180,E1 -25632.354,E2 -25632.354} C_VEL
LIN {X 0,Y 120.492,Z 370.377,A -85,B 0,C 180,E1 -25636.508,E2 -25636.508} C_VEL
LIN {X 0,Y 119.81,Z 375.116,A -85,B 0,C 180,E1 -25641.567,E2 -25641.567} C_VEL
LIN {X 0,Y 119.793,Z 378.673,A -85,B 0,C 180,E1 -25646.637,E2 -25646.637} C_VEL
LIN {X 0,Y 119.963,Z 380.446,A -85,B 0,C 180,E1 -25650,E2 -25650} C_VEL
LIN {X 0,Y 119.684,Z 381.68,A -85,B 0,C 180,E1 -25653.366,E2 -25653.366} C_VEL
LIN {X 0,Y 119.783,Z 382.965,A -85,B 0,C 180,E1 -25660.138,E2 -25660.138} C_VEL
LIN {X 0,Y 120.398,Z 383.05,A -85,B 0,C 180,E1 -25663.503,E2 -25663.503} C_VEL
LIN {X 0,Y 122.826,Z 382.042,A -85,B 0,C 180,E1 -25670.079,E2 -25670.079} C_VEL
LIN {X 0,Y 126.978,Z 379.551,A -85,B 0,C 180,E1 -25676.281,E2 -25676.281} C_VEL
LIN {X 0,Y 131.39,Z 376.379,A -85,B 0,C 180,E1 -25680.947,E2 -25680.947} C_VEL
LIN {X 0,Y 137.573,Z 371.252,A -85,B 0,C 180,E1 -25685.978,E2 -25685.978} C_VEL
LIN {X 0,Y 142.031,Z 367.189,A -85,B 0,C 180,E1 -25688.836,E2 -25688.836} C_VEL
LIN {X 0,Y 144.534,Z 364.405,A -85,B 0,C 180,E1 -25690.659,E2 -25690.659} C_VEL
LIN {X 0,Y 147.471,Z 359.614,A -85,B 0,C 180,E1 -25693.86,E2 -25693.86} C_VEL
LIN {X 0,Y 150.592,Z 354.334,A -85,B 0,C 180,E1 -25696.838,E2 -25696.838} C_VEL
LIN {X 0,Y 153.279,Z 350.716,A -85,B 0,C 180,E1 -25698.278,E2 -25698.278} C_VEL
LIN {X 0,Y 160.846,Z 341.03,A -85,B 0,C 180,E1 -25700.856,E2 -25700.856} C_VEL
LIN {X 0,Y 167.594,Z 330.8,A -85,B 0,C 180,E1 -25702.821,E2 -25702.821} C_VEL
LIN {X 0,Y 173.846,Z 319.452,A -85,B 0,C 180,E1 -25704.447,E2 -25704.447} C_VEL
LIN {X 0,Y 178.923,Z 308.332,A -85,B 0,C 180,E1 -25705.574,E2 -25705.574} C_VEL
LIN {X 0,Y 183.418,Z 295.589,A -85,B 0,C 180,E1 -25706.53,E2 -25706.53} C_VEL
LIN {X 0,Y 186.935,Z 281.875,A -85,B 0,C 180,E1 -25707.25,E2 -25707.25} C_VEL
LIN {X 0,Y 189.164,Z 267.433,A -85,B 0,C 180,E1 -25707.763,E2 -25707.763} C_VEL
LIN {X 0,Y 189.539,Z 264.003,A -85,B 0,C 180,E1 -25707.908,E2 -25707.908} C_VEL
LIN {X 0,Y 188.093,Z 258.333,A -85,B 0,C 180,E1 -25710.392,E2 -25710.392} C_VEL
LIN {X 0,Y 187.075,Z 254.852,A -85,B 0,C 180,E1 -25712.365,E2 -25712.365} C_VEL
LIN {X 0,Y 186.273,Z 252.028,A -85,B 0,C 180,E1 -25714.395,E2 -25714.395} C_VEL
LIN {X 0,Y 185.359,Z 248.617,A -85,B 0,C 180,E1 -25717.718,E2 -25717.718} C_VEL
LIN {X 0,Y 185.019,Z 247.193,A -85,B 0,C 180,E1 -25720.687,E2 -25720.687} C_VEL
LIN {X 0,Y 185.414,Z 247.264,A -85,B 0,C 180,E1 -25725.59,E2 -25725.59} C_VEL
LIN {X 0,Y 185.623,Z 247.874,A -85,B 0,C 180,E1 -25726.684,E2 -25726.684} C_VEL
LIN {X 0,Y 187.523,Z 251.77,A -85,B 0,C 180,E1 -25731.538,E2 -25731.538} C_VEL
LIN {X 0,Y 188.626,Z 254.588,A -85,B 0,C 180,E1 -25733.486,E2 -25733.486} C_VEL
LIN {X 0,Y 190.125,Z 258.193,A -85,B 0,C 180,E1 -25735.698,E2 -25735.698} C_VEL
LIN {X 0,Y 187.759,Z 274.953,A -85,B 0,C 180,E1 -25736.378,E2 -25736.378} C_VEL
LIN {X 0,Y 184.624,Z 288.015,A -85,B 0,C 180,E1 -25737.165,E2 -25737.165} C_VEL
LIN {X 0,Y 180.613,Z 300.276,A -85,B 0,C 180,E1 -25738.265,E2 -25738.265} C_VEL
LIN {X 0,Y 175.702,Z 311.885,A -85,B 0,C 180,E1 -25739.657,E2 -25739.657} C_VEL
LIN {X 0,Y 169.604,Z 323.268,A -85,B 0,C 180,E1 -25741.462,E2 -25741.462} C_VEL
LIN {X 0,Y 163.514,Z 332.71,A -85,B 0,C 180,E1 -25743.432,E2 -25743.432} C_VEL
LIN {X 0,Y 156.804,Z 341.588,A -85,B 0,C 180,E1 -25745.909,E2 -25745.909} C_VEL
LIN {X 0,Y 149.423,Z 349.794,A -85,B 0,C 180,E1 -25748.991,E2 -25748.991} C_VEL
LIN {X 0,Y 142.179,Z 356.664,A -85,B 0,C 180,E1 -25752.516,E2 -25752.516} C_VEL
LIN {X 0,Y 135.556,Z 362.052,A -85,B 0,C 180,E1 -25756.436,E2 -25756.436} C_VEL
LIN {X 0,Y 130.436,Z 365.572,A -85,B 0,C 180,E1 -25760.057,E2 -25760.057} C_VEL
LIN {X 0,Y 124.475,Z 368.997,A -85,B 0,C 180,E1 -25765.396,E2 -25765.396} C_VEL
LIN {X 0,Y 120.953,Z 370.509,A -85,B 0,C 180,E1 -25769.358,E2 -25769.358} C_VEL
LIN {X 0,Y 118.031,Z 371.373,A -85,B 0,C 180,E1 -25773.529,E2 -25773.529} C_VEL
LIN {X 0,Y 115.726,Z 371.6,A -85,B 0,C 180,E1 -25777.864,E2 -25777.864} C_VEL
LIN {X 0,Y 113.777,Z 371.077,A -85,B 0,C 180,E1 -25782.801,E2 -25782.801} C_VEL
LIN {X 0,Y 112.508,Z 369.538,A -85,B 0,C 180,E1 -25788.554,E2 -25788.554} C_VEL
LIN {X 0,Y 112.248,Z 366.21,A -85,B 0,C 180,E1 -25795.702,E2 -25795.702} C_VEL
LIN {X 0,Y 112.854,Z 362.861,A -85,B 0,C 180,E1 -25800.674,E2 -25800.674} C_VEL
LIN {X 0,Y 114.115,Z 358.282,A -85,B 0,C 180,E1 -25805.85,E2 -25805.85} C_VEL
LIN {X 0,Y 116.117,Z 351.785,A -85,B 0,C 180,E1 -25811.473,E2 -25811.473} C_VEL
LIN {X 0,Y 118.66,Z 344.565,A -85,B 0,C 180,E1 -25816.296,E2 -25816.296} C_VEL
LIN {X 0,Y 121.886,Z 335.604,A -85,B 0,C 180,E1 -25820.949,E2 -25820.949} C_VEL
LIN {X 0,Y 125.103,Z 326.299,A -85,B 0,C 180,E1 -25824.681,E2 -25824.681} C_VEL
LIN {X 0,Y 128.557,Z 315.432,A -85,B 0,C 180,E1 -25828.042,E2 -25828.042} C_VEL
LIN {X 0,Y 131.575,Z 304.614,A -85,B 0,C 180,E1 -25830.625,E2 -25830.625} C_VEL
LIN {X 0,Y 134.282,Z 293.08,A -85,B 0,C 180,E1 -25832.723,E2 -25832.723} C_VEL
LIN {X 0,Y 136.622,Z 279.529,A -85,B 0,C 180,E1 -25834.518,E2 -25834.518} C_VEL
LIN {X 0,Y 138.33,Z 265.944,A -85,B 0,C 180,E1 -25835.695,E2 -25835.695} C_VEL
LIN {X 0,Y 141.55,Z 223.079,A -85,B 0,C 180,E1 -25837.919,E2 -25837.919} C_VEL
LIN {X 0,Y 135.685,Z 209.021,A -85,B 0,C 180,E1 -25840.683,E2 -25840.683} C_VEL
LIN {X 0,Y 127.162,Z 193.467,A -85,B 0,C 180,E1 -25844.861,E2 -25844.861} C_VEL
LIN {X 0,Y 120.124,Z 182.678,A -85,B 0,C 180,E1 -25848.762,E2 -25848.762} C_VEL
LIN {X 0,Y 117.588,Z 178.834,A -85,B 0,C 180,E1 -25850.313,E2 -25850.313} C_VEL
LIN {X 0,Y 115.645,Z 176.468,A -85,B 0,C 180,E1 -25851.506,E2 -25851.506} C_VEL
LIN {X 0,Y 114.968,Z 174.162,A -85,B 0,C 180,E1 -25852.13,E2 -25852.13} C_VEL
LIN {X 0,Y 114.857,Z 174.177,A -85,B 0,C 180,E1 -25859.309,E2 -25859.309} C_VEL
LIN {X 0,Y 114.814,Z 174.183,A -85,B 0,C 180,E1 -25863.429,E2 -25863.429} C_VEL
LIN {X 0,Y 114.776,Z 174.187,A -85,B 0,C 180,E1 -25867.757,E2 -25867.757} C_VEL
LIN {X 0,Y 114.779,Z 174.174,A -85,B 0,C 180,E1 -25872.713,E2 -25872.713} C_VEL
LIN {X 0,Y 114.8,Z 174.175,A -85,B 0,C 180,E1 -25877.67,E2 -25877.67} C_VEL
LIN {X 0,Y 114.811,Z 174.171,A -85,B 0,C 180,E1 -25882.729,E2 -25882.729} C_VEL
LIN {X 0,Y 114.863,Z 174.156,A -85,B 0,C 180,E1 -25888.937,E2 -25888.937} C_VEL
LIN {X 0,Y 114.946,Z 174.166,A -85,B 0,C 180,E1 -25896.509,E2 -25896.509} C_VEL
LIN {X 0,Y 115.017,Z 174.129,A -85,B 0,C 180,E1 -25902.211,E2 -25902.211} C_VEL
LIN {X 0,Y 115.284,Z 174.123,A -85,B 0,C 180,E1 -25907.263,E2 -25907.263} C_VEL
LIN {X 0,Y 115.388,Z 174.084,A -85,B 0,C 180,E1 -25913.004,E2 -25913.004} C_VEL
LIN {X 0,Y 115.995,Z 174.03,A -85,B 0,C 180,E1 -25920.001,E2 -25920.001} C_VEL
LIN {X 0,Y 115.388,Z 174.106,A -85,B 0,C 180,E1 -25926.998,E2 -25926.998} C_VEL
LIN {X 0,Y 115.285,Z 174.106,A -85,B 0,C 180,E1 -25932.738,E2 -25932.738} C_VEL
LIN {X 0,Y 115.018,Z 174.155,A -85,B 0,C 180,E1 -25937.79,E2 -25937.79} C_VEL
LIN {X 0,Y 114.947,Z 174.167,A -85,B 0,C 180,E1 -25943.492,E2 -25943.492} C_VEL
LIN {X 0,Y 114.891,Z 174.177,A -85,B 0,C 180,E1 -25949.932,E2 -25949.932} C_VEL
LIN {X 0,Y 115.983,Z 177.19,A -85,B 0,C 180,E1 -25950.835,E2 -25950.835} C_VEL
LIN {X 0,Y 118.037,Z 179.582,A -85,B 0,C 180,E1 -25952.08,E2 -25952.08} C_VEL
LIN {X 0,Y 120.019,Z 182.745,A -85,B 0,C 180,E1 -25953.298,E2 -25953.298} C_VEL
LIN {X 0,Y 125.546,Z 191.638,A -85,B 0,C 180,E1 -25956.43,E2 -25956.43} C_VEL
LIN {X 0,Y 130.067,Z 201.636,A -85,B 0,C 180,E1 -25958.945,E2 -25958.945} C_VEL
LIN {X 0,Y 134.914,Z 213.777,A -85,B 0,C 180,E1 -25961.527,E2 -25961.527} C_VEL
LIN {X 0,Y 139.326,Z 226.987,A -85,B 0,C 180,E1 -25963.822,E2 -25963.822} C_VEL
LIN {X 0,Y 140.413,Z 244.531,A -85,B 0,C 180,E1 -25965.367,E2 -25965.367} C_VEL
LIN {X 0,Y 137.532,Z 281.067,A -85,B 0,C 180,E1 -25967.305,E2 -25967.305} C_VEL
LIN {X 0,Y 135.856,Z 293.084,A -85,B 0,C 180,E1 -25968.362,E2 -25968.362} C_VEL
LIN {X 0,Y 133.337,Z 306.025,A -85,B 0,C 180,E1 -25970.03,E2 -25970.03} C_VEL
LIN {X 0,Y 130.293,Z 317.862,A -85,B 0,C 180,E1 -25972.152,E2 -25972.152} C_VEL
LIN {X 0,Y 126.849,Z 329.288,A -85,B 0,C 180,E1 -25974.913,E2 -25974.913} C_VEL
LIN {X 0,Y 123.375,Z 339.647,A -85,B 0,C 180,E1 -25978.202,E2 -25978.202} C_VEL
LIN {X 0,Y 120.092,Z 348.976,A -85,B 0,C 180,E1 -25982.084,E2 -25982.084} C_VEL
LIN {X 0,Y 117.39,Z 356.657,A -85,B 0,C 180,E1 -25986.164,E2 -25986.164} C_VEL
LIN {X 0,Y 114.964,Z 364.172,A -85,B 0,C 180,E1 -25991.28,E2 -25991.28} C_VEL
LIN {X 0,Y 113.226,Z 371.042,A -85,B 0,C 180,E1 -25997.453,E2 -25997.453} C_VEL
LIN {X 0,Y 112.709,Z 375.526,A -85,B 0,C 180,E1 -26002.836,E2 -26002.836} C_VEL
LIN {X 0,Y 112.738,Z 377.855,A -85,B 0,C 180,E1 -26006.426,E2 -26006.426} C_VEL
LIN {X 0,Y 112.899,Z 379.714,A -85,B 0,C 180,E1 -26010,E2 -26010} C_VEL
LIN {X 0,Y 112.603,Z 381.059,A -85,B 0,C 180,E1 -26013.578,E2 -26013.578} C_VEL
LIN {X 0,Y 112.787,Z 382.471,A -85,B 0,C 180,E1 -26020.774,E2 -26020.774} C_VEL
LIN {X 0,Y 114.558,Z 382.404,A -85,B 0,C 180,E1 -26027.863,E2 -26027.863} C_VEL
LIN {X 0,Y 116.17,Z 381.819,A -85,B 0,C 180,E1 -26031.283,E2 -26031.283} C_VEL
LIN {X 0,Y 120.638,Z 379.471,A -85,B 0,C 180,E1 -26037.778,E2 -26037.778} C_VEL
LIN {X 0,Y 126.6,Z 375.6,A -85,B 0,C 180,E1 -26043.72,E2 -26043.72} C_VEL
LIN {X 0,Y 131.904,Z 371.562,A -85,B 0,C 180,E1 -26047.787,E2 -26047.787} C_VEL
LIN {X 0,Y 137.99,Z 366.461,A -85,B 0,C 180,E1 -26051.46,E2 -26051.46} C_VEL
LIN {X 0,Y 145.788,Z 358.949,A -85,B 0,C 180,E1 -26055.32,E2 -26055.32} C_VEL
LIN {X 0,Y 153.279,Z 350.716,A -85,B 0,C 180,E1 -26058.278,E2 -26058.278} C_VEL
LIN {X 0,Y 156.005,Z 346.949,A -85,B 0,C 180,E1 -26059.643,E2 -26059.643} C_VEL
LIN {X 0,Y 159.437,Z 340.655,A -85,B 0,C 180,E1 -26062.148,E2 -26062.148} C_VEL
LIN {X 0,Y 162.906,Z 333.888,A -85,B 0,C 180,E1 -26064.371,E2 -26064.371} C_VEL
LIN {X 0,Y 165.572,Z 329.353,A -85,B 0,C 180,E1 -26065.287,E2 -26065.287} C_VEL
LIN {X 0,Y 171.368,Z 319.071,A -85,B 0,C 180,E1 -26066.678,E2 -26066.678} C_VEL
LIN {X 0,Y 176.58,Z 308.037,A -85,B 0,C 180,E1 -26067.753,E2 -26067.753} C_VEL
LIN {X 0,Y 181.076,Z 295.826,A -85,B 0,C 180,E1 -26068.635,E2 -26068.635} C_VEL
LIN {X 0,Y 184.67,Z 282.514,A -85,B 0,C 180,E1 -26069.316,E2 -26069.316} C_VEL
LIN {X 0,Y 187.026,Z 268.674,A -85,B 0,C 180,E1 -26069.8,E2 -26069.8} C_VEL
LIN {X 0,Y 187.111,Z 267.61,A -85,B 0,C 180,E1 -26069.889,E2 -26069.889} C_VEL
LIN {X 0,Y 185.762,Z 262.005,A -85,B 0,C 180,E1 -26072.692,E2 -26072.692} C_VEL
LIN {X 0,Y 184.9,Z 258.531,A -85,B 0,C 180,E1 -26075.18,E2 -26075.18} C_VEL
LIN {X 0,Y 184.236,Z 255.498,A -85,B 0,C 180,E1 -26078.102,E2 -26078.102} C_VEL
LIN {X 0,Y 183.936,Z 254.165,A -85,B 0,C 180,E1 -26081.252,E2 -26081.252} C_VEL
LIN {X 0,Y 184.407,Z 254.343,A -85,B 0,C 180,E1 -26085.772,E2 -26085.772} C_VEL
LIN {X 0,Y 186.193,Z 258.65,A -85,B 0,C 180,E1 -26091.087,E2 -26091.087} C_VEL
LIN {X 0,Y 187.656,Z 262.63,A -85,B 0,C 180,E1 -26093.785,E2 -26093.785} C_VEL
LIN {X 0,Y 185.378,Z 276.9,A -85,B 0,C 180,E1 -26094.369,E2 -26094.369} C_VEL
LIN {X 0,Y 182.059,Z 289.755,A -85,B 0,C 180,E1 -26095.156,E2 -26095.156} C_VEL
LIN {X 0,Y 177.437,Z 302.823,A -85,B 0,C 180,E1 -26096.334,E2 -26096.334} C_VEL
LIN {X 0,Y 172.027,Z 314.477,A -85,B 0,C 180,E1 -26097.771,E2 -26097.771} C_VEL
LIN {X 0,Y 166.033,Z 324.953,A -85,B 0,C 180,E1 -26099.446,E2 -26099.446} C_VEL
LIN {X 0,Y 159.295,Z 334.751,A -85,B 0,C 180,E1 -26101.505,E2 -26101.505} C_VEL
LIN {X 0,Y 153.167,Z 342.369,A -85,B 0,C 180,E1 -26103.654,E2 -26103.654} C_VEL
LIN {X 0,Y 146.676,Z 349.303,A -85,B 0,C 180,E1 -26106.16,E2 -26106.16} C_VEL
LIN {X 0,Y 139.838,Z 355.609,A -85,B 0,C 180,E1 -26109.21,E2 -26109.21} C_VEL
LIN {X 0,Y 132.38,Z 361.46,A -85,B 0,C 180,E1 -26113.174,E2 -26113.174} C_VEL
LIN {X 0,Y 125.42,Z 366.046,A -85,B 0,C 180,E1 -26117.712,E2 -26117.712} C_VEL
LIN {X 0,Y 120.792,Z 368.557,A -85,B 0,C 180,E1 -26121.422,E2 -26121.422} C_VEL
LIN {X 0,Y 116.711,Z 370.391,A -85,B 0,C 180,E1 -26125.412,E2 -26125.412} C_VEL
LIN {X 0,Y 113.091,Z 371.536,A -85,B 0,C 180,E1 -26129.811,E2 -26129.811} C_VEL
LIN {X 0,Y 109.732,Z 372.011,A -85,B 0,C 180,E1 -26135.198,E2 -26135.198} C_VEL
LIN {X 0,Y 107.183,Z 371.548,A -85,B 0,C 180,E1 -26140.972,E2 -26140.972} C_VEL
LIN {X 0,Y 105.451,Z 369.697,A -85,B 0,C 180,E1 -26148.205,E2 -26148.205} C_VEL
LIN {X 0,Y 105.154,Z 366.307,A -85,B 0,C 180,E1 -26155.584,E2 -26155.584} C_VEL
LIN {X 0,Y 106.053,Z 361.727,A -85,B 0,C 180,E1 -26162.363,E2 -26162.363} C_VEL
LIN {X 0,Y 107.932,Z 355.544,A -85,B 0,C 180,E1 -26169.015,E2 -26169.015} C_VEL
LIN {X 0,Y 110.74,Z 347.618,A -85,B 0,C 180,E1 -26175.294,E2 -26175.294} C_VEL
LIN {X 0,Y 113.681,Z 339.816,A -85,B 0,C 180,E1 -26180.021,E2 -26180.021} C_VEL
LIN {X 0,Y 117.196,Z 330.408,A -85,B 0,C 180,E1 -26184.408,E2 -26184.408} C_VEL
LIN {X 0,Y 120.945,Z 319.39,A -85,B 0,C 180,E1 -26188.335,E2 -26188.335} C_VEL
LIN {X 0,Y 124.189,Z 308.784,A -85,B 0,C 180,E1 -26191.216,E2 -26191.216} C_VEL
LIN {X 0,Y 127.344,Z 296.692,A -85,B 0,C 180,E1 -26193.677,E2 -26193.677} C_VEL
LIN {X 0,Y 129.921,Z 283.795,A -85,B 0,C 180,E1 -26195.627,E2 -26195.627} C_VEL
